  Call Extruder(0.094)
  MoveL 4443 to (501.07, 492.3, 9.5) mm, rotated rx 0 ry 90 rz 0 deg; joints [-11.281, -27.301, 111.303, -15.284, -83.35, 50.807]
  Call Extruder(0.055)
  MoveL 4444 to (501.07, 490.4, 9.5) mm, rotated rx 0 ry 90 rz 0 deg; joints [-11.107, -27.308, 111.347, -15.107, -83.382, 50.779]
  Call Extruder(0.248)
  MoveL 4445 to (509.6, 490.4, 9.5) mm, rotated rx 0 ry 90 rz 0 deg; joints [-10.955, -27.148, 110.323, -14.982, -82.543, 50.989]
  Call Extruder(0.228)
  MoveL 4446 to (509.6, 498.23, 9.5) mm, rotated rx 0 ry 90 rz 0 deg; joints [-11.664, -27.118, 110.135, -15.702, -82.413, 51.114]
  Call Extruder(0.043)
  MoveL 4447 to (508.13, 498.23, 9.5) mm, rotated rx 0 ry 90 rz 0 deg; joints [-11.692, -27.146, 110.312, -15.725, -82.557, 51.076]
  Call Extruder(0.014)
  MoveL 4448 to (507.66, 498.23, 9.5) mm, rotated rx 0 ry 90 rz 0 deg; joints [-11.701, -27.155, 110.368, -15.733, -82.602, 51.065]
  Call Extruder(0.080)
  MoveL 4449 to (507.66, 500.97, 9.5) mm, rotated rx 0 ry 90 rz 0 deg; joints [-11.949, -27.144, 110.299, -15.985, -82.555, 51.109]
  Set speed (120.0 mm/s)
  MoveL 4450 to (508.06, 500.97, 9.5) mm, rotated rx 0 ry 90 rz 0 deg; joints [-11.941, -27.137, 110.251, -15.978, -82.516, 51.119]
  Set speed (1000.0 mm/s)
  MoveL 4451 to (508.06, 501.67, 9.5) mm, rotated rx 0 ry 90 rz 0 deg; joints [-12.005, -27.134, 110.233, -16.043, -82.504, 51.131]
  Set speed (1000.0 mm/s)
  MoveL 4452 to (490.68, 490.68, 9.5) mm, rotated rx 0 ry 90 rz 0 deg; joints [-11.324, -27.485, 112.575, -15.296, -84.401, 50.522]
  Set speed (1000.0 mm/s)
  MoveL 4453 to (490.68, 490.68, 9.6) mm, rotated rx 0 ry 90 rz 0 deg; joints [-11.324, -27.496, 112.58, -15.296, -84.396, 50.523]
  Set speed (30.0 mm/s)
  Call Extruder(0.767)
  MoveL 4454 to (509.32, 509.32, 9.6) mm, rotated rx 0 ry 90 rz 0 deg; joints [-12.669, -27.086, 109.886, -16.723, -82.239, 51.295]
  MoveL 4455 to (509.44, 509.44, 9.6) mm, rotated rx 0 ry 90 rz 0 deg; joints [-12.677, -27.083, 109.868, -16.733, -82.225, 51.301]
  Set speed (120.0 mm/s)
  MoveL 4456 to (508.59, 501.31, 9.6) mm, rotated rx 0 ry 90 rz 0 deg; joints [-11.962, -27.135, 110.184, -16.001, -82.453, 51.14]
  Set speed (30.0 mm/s)
  Call Extruder(0.330)
  MoveL 4457 to (500.58, 509.32, 9.6) mm, rotated rx 0 ry 90 rz 0 deg; joints [-12.847, -27.254, 110.932, -16.871, -83.085, 51.06]
  Set speed (120.0 mm/s)
  MoveL 4458 to (499.42, 509.32, 9.6) mm, rotated rx 0 ry 90 rz 0 deg; joints [-12.872, -27.276, 111.07, -16.891, -83.198, 51.028]
  Set speed (30.0 mm/s)
  Call Extruder(0.360)
  MoveL 4459 to (490.68, 500.58, 9.6) mm, rotated rx 0 ry 90 rz 0 deg; joints [-12.247, -27.462, 112.336, -16.229, -84.216, 50.659]
  Set speed (120.0 mm/s)
  MoveL 4460 to (490.68, 499.42, 9.6) mm, rotated rx 0 ry 90 rz 0 deg; joints [-12.139, -27.466, 112.366, -16.12, -84.237, 50.642]
  Set speed (30.0 mm/s)
  Call Extruder(0.286)
  MoveL 4461 to (497.63, 492.47, 9.6) mm, rotated rx 0 ry 90 rz 0 deg; joints [-11.361, -27.372, 111.714, -15.354, -83.68, 50.724]
  MoveL 4462 to (497.75, 492.35, 9.6) mm, rotated rx 0 ry 90 rz 0 deg; joints [-11.347, -27.371, 111.702, -15.34, -83.67, 50.726]
  Set speed (120.0 mm/s)
  MoveL 4463 to (501.03, 492.33, 9.6) mm, rotated rx 0 ry 90 rz 0 deg; joints [-11.285, -27.312, 111.312, -15.287, -83.348, 50.808]
  Set speed (1000.0 mm/s)
  MoveL 4464 to (501.28, 491.38, 9.6) mm, rotated rx 0 ry 90 rz 0 deg; joints [-11.193, -27.311, 111.304, -15.196, -83.339, 50.8]
  Set speed (30.0 mm/s)
  Call Extruder(0.268)
  MoveL 4465 to (507.79, 497.89, 9.6) mm, rotated rx 0 ry 90 rz 0 deg; joints [-11.668, -27.165, 110.366, -15.699, -82.59, 51.064]
  MoveL 4466 to (507.91, 498.02, 9.6) mm, rotated rx 0 ry 90 rz 0 deg; joints [-11.676, -27.162, 110.348, -15.709, -82.576, 51.069]
  Set speed (120.0 mm/s)
  MoveL 4467 to (509.32, 490.68, 9.6) mm, rotated rx 0 ry 90 rz 0 deg; joints [-10.985, -27.163, 110.356, -15.012, -82.561, 50.987]
  Set speed (30.0 mm/s)
  Call Extruder(0.767)
  MoveL 4468 to (490.68, 509.32, 9.6) mm, rotated rx 0 ry 90 rz 0 deg; joints [-13.056, -27.429, 112.105, -17.048, -84.046, 50.787]
  MoveL 4469 to (490.56, 509.44, 9.6) mm, rotated rx 0 ry 90 rz 0 deg; joints [-13.07, -27.431, 112.116, -17.062, -84.056, 50.785]
  Set speed (120.0 mm/s)
  MoveL 4470 to (507.59, 501.1, 9.6) mm, rotated rx 0 ry 90 rz 0 deg; joints [-11.962, -27.156, 110.31, -15.997, -82.554, 51.111]
  Set speed (1000.0 mm/s)
  MoveL 4471 to (507.66, 501.03, 9.6) mm, rotated rx 0 ry 90 rz 0 deg; joints [-11.954, -27.155, 110.303, -15.99, -82.549, 51.111]
  Set speed (15.0 mm/s)
  Call Extruder(0.056)
  MoveL 4472 to (509.6, 501.03, 9.6) mm, rotated rx 0 ry 90 rz 0 deg; joints [-11.917, -27.117, 110.069, -15.96, -82.36, 51.161]
  Call Extruder(0.249)
  MoveL 4473 to (509.6, 509.6, 9.6) mm, rotated rx 0 ry 90 rz 0 deg; joints [-12.688, -27.079, 109.845, -16.744, -82.206, 51.308]
  Call Extruder(0.559)
  MoveL 4474 to (490.4, 509.6, 9.6) mm, rotated rx 0 ry 90 rz 0 deg; joints [-13.088, -27.433, 112.13, -17.079, -84.068, 50.783]
  MoveL 4475 to (490.4, 490.4, 9.6) mm, rotated rx 0 ry 90 rz 0 deg; joints [-11.303, -27.501, 112.62, -15.274, -84.428, 50.513]
  Call Extruder(0.218)
  MoveL 4476 to (497.9, 490.4, 9.6) mm, rotated rx 0 ry 90 rz 0 deg; joints [-11.164, -27.375, 111.731, -15.156, -83.688, 50.702]
  Call Extruder(0.039)
  MoveL 4477 to (497.9, 491.75, 9.6) mm, rotated rx 0 ry 90 rz 0 deg; joints [-11.289, -27.37, 111.699, -15.282, -83.666, 50.721]
  Call Extruder(0.016)
  MoveL 4478 to (497.91, 492.3, 9.6) mm, rotated rx 0 ry 90 rz 0 deg; joints [-11.34, -27.368, 111.685, -15.333, -83.655, 50.729]
  Call Extruder(0.090)
  MoveL 4479 to (501, 492.3, 9.6) mm, rotated rx 0 ry 90 rz 0 deg; joints [-11.283, -27.313, 111.316, -15.285, -83.351, 50.807]
  Call Extruder(0.055)
  MoveL 4480 to (501.01, 490.4, 9.6) mm, rotated rx 0 ry 90 rz 0 deg; joints [-11.108, -27.32, 111.36, -15.108, -83.383, 50.779]
  Call Extruder(0.250)
  MoveL 4481 to (509.6, 490.4, 9.6) mm, rotated rx 0 ry 90 rz 0 deg; joints [-10.955, -27.159, 110.329, -14.982, -82.538, 50.99]
  Call Extruder(0.226)
  MoveL 4482 to (509.6, 498.17, 9.6) mm, rotated rx 0 ry 90 rz 0 deg; joints [-11.659, -27.128, 110.141, -15.697, -82.409, 51.114]
  Call Extruder(0.056)
  MoveL 4483 to (507.66, 498.17, 9.6) mm, rotated rx 0 ry 90 rz 0 deg; joints [-11.695, -27.166, 110.374, -15.727, -82.598, 51.065]
  Call Extruder(0.083)
  MoveL 4484 to (507.66, 501.03, 9.6) mm, rotated rx 0 ry 90 rz 0 deg; joints [-11.954, -27.155, 110.303, -15.99, -82.549, 51.111]
  Set speed (120.0 mm/s)
  MoveL 4485 to (508.06, 501.03, 9.6) mm, rotated rx 0 ry 90 rz 0 deg; joints [-11.947, -27.147, 110.255, -15.984, -82.51, 51.122]
  Set speed (1000.0 mm/s)
  MoveL 4486 to (508.06, 501.73, 9.6) mm, rotated rx 0 ry 90 rz 0 deg; joints [-12.01, -27.144, 110.237, -16.048, -82.497, 51.133]
  Set speed (1000.0 mm/s)
  MoveL 4487 to (490.68, 490.68, 9.6) mm, rotated rx 0 ry 90 rz 0 deg; joints [-11.324, -27.496, 112.58, -15.296, -84.396, 50.523]
  Set speed (1000.0 mm/s)
  MoveL 4488 to (490.68, 490.68, 9.7) mm, rotated rx 0 ry 90 rz 0 deg; joints [-11.324, -27.506, 112.585, -15.296, -84.391, 50.525]
  Set speed (30.0 mm/s)
  Call Extruder(0.767)
  MoveL 4489 to (509.32, 509.32, 9.7) mm, rotated rx 0 ry 90 rz 0 deg; joints [-12.669, -27.097, 109.891, -16.724, -82.234, 51.297]
  MoveL 4490 to (509.44, 509.44, 9.7) mm, rotated rx 0 ry 90 rz 0 deg; joints [-12.677, -27.094, 109.873, -16.733, -82.22, 51.302]
  Set speed (120.0 mm/s)
  MoveL 4491 to (508.53, 501.37, 9.7) mm, rotated rx 0 ry 90 rz 0 deg; joints [-11.968, -27.147, 110.195, -16.007, -82.453, 51.141]
  Set speed (30.0 mm/s)
  Call Extruder(0.327)
  MoveL 4492 to (500.58, 509.32, 9.7) mm, rotated rx 0 ry 90 rz 0 deg; joints [-12.847, -27.265, 110.937, -16.871, -83.08, 51.061]
  Set speed (120.0 mm/s)
  MoveL 4493 to (499.42, 509.32, 9.7) mm, rotated rx 0 ry 90 rz 0 deg; joints [-12.872, -27.286, 111.075, -16.891, -83.193, 51.03]
  Set speed (30.0 mm/s)
  Call Extruder(0.360)
  MoveL 4494 to (490.68, 500.58, 9.7) mm, rotated rx 0 ry 90 rz 0 deg; joints [-12.247, -27.472, 112.342, -16.229, -84.21, 50.66]
  Set speed (120.0 mm/s)
  MoveL 4495 to (490.68, 499.42, 9.7) mm, rotated rx 0 ry 90 rz 0 deg; joints [-12.139, -27.477, 112.371, -16.12, -84.232, 50.644]
  Set speed (30.0 mm/s)
  Call Extruder(0.288)
  MoveL 4496 to (497.68, 492.42, 9.7) mm, rotated rx 0 ry 90 rz 0 deg; joints [-11.355, -27.382, 111.714, -15.348, -83.671, 50.726]
  MoveL 4497 to (497.8, 492.3, 9.7) mm, rotated rx 0 ry 90 rz 0 deg; joints [-11.342, -27.381, 111.703, -15.335, -83.661, 50.728]
  Set speed (120.0 mm/s)
  MoveL 4498 to (500.97, 492.33, 9.7) mm, rotated rx 0 ry 90 rz 0 deg; joints [-11.286, -27.324, 111.324, -15.289, -83.349, 50.808]
  Set speed (1000.0 mm/s)
  MoveL 4499 to (501.22, 491.32, 9.7) mm, rotated rx 0 ry 90 rz 0 deg; joints [-11.189, -27.323, 111.318, -15.191, -83.341, 50.799]
  Set speed (30.0 mm/s)
  Call Extruder(0.268)
  MoveL 4500 to (507.73, 497.83, 9.7) mm, rotated rx 0 ry 90 rz 0 deg; joints [-11.663, -27.177, 110.38, -15.695, -82.592, 51.063]
  MoveL 4501 to (507.85, 497.95, 9.7) mm, rotated rx 0 ry 90 rz 0 deg; joints [-11.672, -27.174, 110.362, -15.704, -82.578, 51.068]
  Set speed (120.0 mm/s)
  MoveL 4502 to (509.32, 490.68, 9.7) mm, rotated rx 0 ry 90 rz 0 deg; joints [-10.985, -27.174, 110.361, -15.012, -82.556, 50.989]
  Set speed (30.0 mm/s)
  Call Extruder(0.767)
  MoveL 4503 to (490.68, 509.32, 9.7) mm, rotated rx 0 ry 90 rz 0 deg; joints [-13.056, -27.44, 112.11, -17.048, -84.041, 50.789]
  MoveL 4504 to (490.56, 509.44, 9.7) mm, rotated rx 0 ry 90 rz 0 deg; joints [-13.07, -27.441, 112.121, -17.062, -84.051, 50.787]
  Set speed (120.0 mm/s)
  MoveL 4505 to (501.01, 492.37, 9.7) mm, rotated rx 0 ry 90 rz 0 deg; joints [-11.289, -27.323, 111.318, -15.292, -83.344, 50.809]
  Set speed (1000.0 mm/s)
  MoveL 4506 to (500.94, 492.3, 9.7) mm, rotated rx 0 ry 90 rz 0 deg; joints [-11.284, -27.325, 111.328, -15.286, -83.352, 50.806]
  Set speed (15.0 mm/s)
  Call Extruder(0.055)
  MoveL 4507 to (500.94, 490.4, 9.7) mm, rotated rx 0 ry 90 rz 0 deg; joints [-11.109, -27.332, 111.373, -15.109, -83.384, 50.779]
  Call Extruder(0.252)
  MoveL 4508 to (509.6, 490.4, 9.7) mm, rotated rx 0 ry 90 rz 0 deg; joints [-10.955, -27.169, 110.334, -14.982, -82.533, 50.991]
  Call Extruder(0.224)
  MoveL 4509 to (509.6, 498.11, 9.7) mm, rotated rx 0 ry 90 rz 0 deg; joints [-11.653, -27.139, 110.148, -15.692, -82.405, 51.115]
  Call Extruder(0.056)
  MoveL 4510 to (507.66, 498.11, 9.7) mm, rotated rx 0 ry 90 rz 0 deg; joints [-11.69, -27.177, 110.381, -15.722, -82.594, 51.066]
  Call Extruder(0.087)
  MoveL 4511 to (507.66, 501.09, 9.7) mm, rotated rx 0 ry 90 rz 0 deg; joints [-11.959, -27.165, 110.306, -15.995, -82.542, 51.114]
  Call Extruder(0.056)
  MoveL 4512 to (509.6, 501.09, 9.7) mm, rotated rx 0 ry 90 rz 0 deg; joints [-11.923, -27.127, 110.073, -15.965, -82.353, 51.164]
  Call Extruder(0.248)
  MoveL 4513 to (509.6, 509.6, 9.7) mm, rotated rx 0 ry 90 rz 0 deg; joints [-12.688, -27.09, 109.85, -16.745, -82.201, 51.309]
  Call Extruder(0.559)
  MoveL 4514 to (490.4, 509.6, 9.7) mm, rotated rx 0 ry 90 rz 0 deg; joints [-13.088, -27.443, 112.135, -17.079, -84.063, 50.785]
  MoveL 4515 to (490.4, 490.4, 9.7) mm, rotated rx 0 ry 90 rz 0 deg; joints [-11.303, -27.512, 112.625, -15.274, -84.423, 50.514]
  Call Extruder(0.220)
  MoveL 4516 to (497.95, 490.4, 9.7) mm, rotated rx 0 ry 90 rz 0 deg; joints [-11.163, -27.385, 111.729, -15.155, -83.678, 50.704]
  Call Extruder(0.055)
  MoveL 4517 to (497.96, 492.3, 9.7) mm, rotated rx 0 ry 90 rz 0 deg; joints [-11.339, -27.378, 111.684, -15.332, -83.645, 50.732]
  Call Extruder(0.087)
  MoveL 4518 to (500.94, 492.3, 9.7) mm, rotated rx 0 ry 90 rz 0 deg; joints [-11.284, -27.325, 111.328, -15.286, -83.352, 50.806]
  Set speed (120.0 mm/s)
  MoveL 4519 to (500.94, 491.9, 9.7) mm, rotated rx 0 ry 90 rz 0 deg; joints [-11.247, -27.326, 111.338, -15.249, -83.359, 50.801]
  Set speed (1000.0 mm/s)
  MoveL 4520 to (501.64, 491.9, 9.7) mm, rotated rx 0 ry 90 rz 0 deg; joints [-11.234, -27.314, 111.254, -15.238, -83.29, 50.818]
  Set speed (1000.0 mm/s)
  MoveL 4521 to (497.93, 492.32, 9.7) mm, rotated rx 0 ry 90 rz 0 deg; joints [-11.342, -27.378, 111.686, -15.336, -83.647, 50.731]
  Set speed (1000.0 mm/s)
  MoveL 4522 to (490.68, 490.68, 9.7) mm, rotated rx 0 ry 90 rz 0 deg; joints [-11.324, -27.506, 112.585, -15.296, -84.391, 50.525]
  Set speed (1000.0 mm/s)
  MoveL 4523 to (490.68, 490.68, 9.8) mm, rotated rx 0 ry 90 rz 0 deg; joints [-11.324, -27.517, 112.591, -15.296, -84.385, 50.526]
  Set speed (30.0 mm/s)
  Call Extruder(0.767)
  MoveL 4524 to (509.32, 509.32, 9.8) mm, rotated rx 0 ry 90 rz 0 deg; joints [-12.669, -27.107, 109.896, -16.724, -82.229, 51.298]
  MoveL 4525 to (509.44, 509.44, 9.8) mm, rotated rx 0 ry 90 rz 0 deg; joints [-12.677, -27.104, 109.878, -16.733, -82.214, 51.304]
  Set speed (120.0 mm/s)
  MoveL 4526 to (508.47, 501.42, 9.8) mm, rotated rx 0 ry 90 rz 0 deg; joints [-11.974, -27.158, 110.205, -16.014, -82.452, 51.142]
  Set speed (30.0 mm/s)
  Call Extruder(0.325)
  MoveL 4527 to (500.58, 509.32, 9.8) mm, rotated rx 0 ry 90 rz 0 deg; joints [-12.847, -27.275, 110.943, -16.871, -83.075, 51.063]
  Set speed (120.0 mm/s)
  MoveL 4528 to (499.42, 509.32, 9.8) mm, rotated rx 0 ry 90 rz 0 deg; joints [-12.872, -27.297, 111.081, -16.891, -83.188, 51.031]
  Set speed (30.0 mm/s)
  Call Extruder(0.360)
  MoveL 4529 to (490.68, 500.58, 9.8) mm, rotated rx 0 ry 90 rz 0 deg; joints [-12.247, -27.483, 112.347, -16.229, -84.205, 50.662]
  Set speed (120.0 mm/s)
  MoveL 4530 to (490.68, 499.42, 9.8) mm, rotated rx 0 ry 90 rz 0 deg; joints [-12.139, -27.487, 112.376, -16.12, -84.227, 50.645]
  Set speed (30.0 mm/s)
  Call Extruder(0.290)
  MoveL 4531 to (497.73, 492.36, 9.8) mm, rotated rx 0 ry 90 rz 0 deg; joints [-11.349, -27.392, 111.714, -15.342, -83.661, 50.728]
  MoveL 4532 to (497.86, 492.24, 9.8) mm, rotated rx 0 ry 90 rz 0 deg; joints [-11.335, -27.39, 111.702, -15.329, -83.651, 50.73]
  Set speed (120.0 mm/s)
  MoveL 4533 to (500.9, 492.32, 9.8) mm, rotated rx 0 ry 90 rz 0 deg; joints [-11.287, -27.336, 111.337, -15.29, -83.35, 50.807]
  Set speed (1000.0 mm/s)
  MoveL 4534 to (501.16, 491.26, 9.8) mm, rotated rx 0 ry 90 rz 0 deg; joints [-11.184, -27.335, 111.332, -15.186, -83.343, 50.798]
  Set speed (30.0 mm/s)
  Call Extruder(0.268)
  MoveL 4535 to (507.67, 497.77, 9.8) mm, rotated rx 0 ry 90 rz 0 deg; joints [-11.659, -27.189, 110.394, -15.69, -82.594, 51.062]
  MoveL 4536 to (507.79, 497.89, 9.8) mm, rotated rx 0 ry 90 rz 0 deg; joints [-11.668, -27.186, 110.376, -15.7, -82.58, 51.067]
  Set speed (120.0 mm/s)
  MoveL 4537 to (509.32, 490.68, 9.8) mm, rotated rx 0 ry 90 rz 0 deg; joints [-10.985, -27.184, 110.366, -15.012, -82.55, 50.99]
  Set speed (30.0 mm/s)
  Call Extruder(0.767)
  MoveL 4538 to (490.68, 509.32, 9.8) mm, rotated rx 0 ry 90 rz 0 deg; joints [-13.056, -27.45, 112.115, -17.048, -84.036, 50.79]
  MoveL 4539 to (490.56, 509.44, 9.8) mm, rotated rx 0 ry 90 rz 0 deg; joints [-13.07, -27.452, 112.127, -17.062, -84.046, 50.789]
  Set speed (120.0 mm/s)
  MoveL 4540 to (500.95, 492.37, 9.8) mm, rotated rx 0 ry 90 rz 0 deg; joints [-11.29, -27.335, 111.331, -15.293, -83.345, 50.809]
  Set speed (1000.0 mm/s)
  MoveL 4541 to (500.88, 492.3, 9.8) mm, rotated rx 0 ry 90 rz 0 deg; joints [-11.285, -27.336, 111.341, -15.287, -83.353, 50.806]
  Set speed (15.0 mm/s)
  Call Extruder(0.055)
  MoveL 4542 to (500.88, 490.4, 9.8) mm, rotated rx 0 ry 90 rz 0 deg; joints [-11.11, -27.343, 111.386, -15.111, -83.385, 50.779]
  Call Extruder(0.254)
  MoveL 4543 to (509.6, 490.4, 9.8) mm, rotated rx 0 ry 90 rz 0 deg; joints [-10.955, -27.18, 110.339, -14.982, -82.527, 50.993]
  Call Extruder(0.223)
  MoveL 4544 to (509.6, 498.05, 9.8) mm, rotated rx 0 ry 90 rz 0 deg; joints [-11.648, -27.15, 110.155, -15.686, -82.401, 51.115]
  Call Extruder(0.056)
  MoveL 4545 to (507.66, 498.05, 9.8) mm, rotated rx 0 ry 90 rz 0 deg; joints [-11.684, -27.188, 110.388, -15.716, -82.59, 51.066]
  Call Extruder(0.090)
  MoveL 4546 to (507.66, 501.14, 9.8) mm, rotated rx 0 ry 90 rz 0 deg; joints [-11.964, -27.175, 110.31, -16.001, -82.536, 51.116]
  Call Extruder(0.056)
  MoveL 4547 to (509.6, 501.15, 9.8) mm, rotated rx 0 ry 90 rz 0 deg; joints [-11.928, -27.137, 110.077, -15.971, -82.347, 51.166]
  Call Extruder(0.246)
  MoveL 4548 to (509.6, 509.6, 9.8) mm, rotated rx 0 ry 90 rz 0 deg; joints [-12.688, -27.1, 109.855, -16.745, -82.196, 51.311]
  Call Extruder(0.559)
  MoveL 4549 to (490.4, 509.6, 9.8) mm, rotated rx 0 ry 90 rz 0 deg; joints [-13.088, -27.454, 112.141, -17.08, -84.058, 50.787]
  MoveL 4550 to (490.4, 490.4, 9.8) mm, rotated rx 0 ry 90 rz 0 deg; joints [-11.303, -27.522, 112.63, -15.274, -84.418, 50.515]
  Call Extruder(0.221)
  MoveL 4551 to (498.01, 490.4, 9.8) mm, rotated rx 0 ry 90 rz 0 deg; joints [-11.162, -27.394, 111.728, -15.154, -83.667, 50.707]
  Call Extruder(0.055)
  MoveL 4552 to (498.02, 492.3, 9.8) mm, rotated rx 0 ry 90 rz 0 deg; joints [-11.338, -27.387, 111.682, -15.332, -83.634, 50.734]
  Call Extruder(0.083)
  MoveL 4553 to (500.88, 492.3, 9.8) mm, rotated rx 0 ry 90 rz 0 deg; joints [-11.285, -27.336, 111.341, -15.287, -83.353, 50.806]
  Set speed (120.0 mm/s)
  MoveL 4554 to (500.88, 491.9, 9.8) mm, rotated rx 0 ry 90 rz 0 deg; joints [-11.248, -27.338, 111.351, -15.25, -83.36, 50.8]
  Set speed (1000.0 mm/s)
  MoveL 4555 to (501.58, 491.9, 9.8) mm, rotated rx 0 ry 90 rz 0 deg; joints [-11.235, -27.325, 111.267, -15.239, -83.291, 50.818]
  Set speed (1000.0 mm/s)
  MoveL 4556 to (497.99, 492.33, 9.8) mm, rotated rx 0 ry 90 rz 0 deg; joints [-11.341, -27.388, 111.685, -15.335, -83.636, 50.734]
  Set speed (1000.0 mm/s)
  MoveL 4557 to (490.68, 490.68, 9.8) mm, rotated rx 0 ry 90 rz 0 deg; joints [-11.324, -27.517, 112.591, -15.296, -84.385, 50.526]
  Set speed (1000.0 mm/s)
  MoveL 4558 to (490.68, 490.68, 9.9) mm, rotated rx 0 ry 90 rz 0 deg; joints [-11.324, -27.528, 112.596, -15.296, -84.38, 50.528]
  Set speed (30.0 mm/s)
  Call Extruder(0.767)
  MoveL 4559 to (509.32, 509.32, 9.9) mm, rotated rx 0 ry 90 rz 0 deg; joints [-12.669, -27.118, 109.902, -16.724, -82.224, 51.3]
  MoveL 4560 to (509.44, 509.44, 9.9) mm, rotated rx 0 ry 90 rz 0 deg; joints [-12.677, -27.115, 109.883, -16.733, -82.209, 51.305]
  Set speed (120.0 mm/s)
  MoveL 4561 to (508.42, 501.48, 9.9) mm, rotated rx 0 ry 90 rz 0 deg; joints [-11.98, -27.169, 110.216, -16.02, -82.452, 51.143]
  Set speed (30.0 mm/s)
  Call Extruder(0.323)
  MoveL 4562 to (500.58, 509.32, 9.9) mm, rotated rx 0 ry 90 rz 0 deg; joints [-12.847, -27.286, 110.948, -16.871, -83.07, 51.064]
  Set speed (120.0 mm/s)
  MoveL 4563 to (499.42, 509.32, 9.9) mm, rotated rx 0 ry 90 rz 0 deg; joints [-12.872, -27.307, 111.086, -16.892, -83.183, 51.033]
  Set speed (30.0 mm/s)
  Call Extruder(0.360)
  MoveL 4564 to (490.68, 500.58, 9.9) mm, rotated rx 0 ry 90 rz 0 deg; joints [-12.247, -27.494, 112.352, -16.229, -84.2, 50.663]
  Set speed (120.0 mm/s)
  MoveL 4565 to (490.68, 499.42, 9.9) mm, rotated rx 0 ry 90 rz 0 deg; joints [-12.139, -27.498, 112.382, -16.12, -84.222, 50.647]
  Set speed (30.0 mm/s)
  Call Extruder(0.293)
  MoveL 4566 to (497.79, 492.31, 9.9) mm, rotated rx 0 ry 90 rz 0 deg; joints [-11.343, -27.402, 111.714, -15.336, -83.651, 50.73]
  MoveL 4567 to (497.91, 492.18, 9.9) mm, rotated rx 0 ry 90 rz 0 deg; joints [-11.329, -27.4, 111.702, -15.323, -83.641, 50.732]
  Set speed (120.0 mm/s)
  MoveL 4568 to (500.84, 492.32, 9.9) mm, rotated rx 0 ry 90 rz 0 deg; joints [-11.288, -27.348, 111.35, -15.291, -83.351, 50.807]
  Set speed (1000.0 mm/s)
  MoveL 4569 to (501.09, 491.19, 9.9) mm, rotated rx 0 ry 90 rz 0 deg; joints [-11.179, -27.347, 111.347, -15.181, -83.345, 50.797]
  Set speed (30.0 mm/s)
  Call Extruder(0.268)
  MoveL 4570 to (507.61, 497.71, 9.9) mm, rotated rx 0 ry 90 rz 0 deg; joints [-11.654, -27.2, 110.408, -15.686, -82.596, 51.061]
  MoveL 4571 to (507.73, 497.83, 9.9) mm, rotated rx 0 ry 90 rz 0 deg; joints [-11.663, -27.198, 110.39, -15.695, -82.582, 51.066]
  Set speed (120.0 mm/s)
  MoveL 4572 to (509.32, 490.68, 9.9) mm, rotated rx 0 ry 90 rz 0 deg; joints [-10.985, -27.195, 110.372, -15.012, -82.545, 50.992]
  Set speed (30.0 mm/s)
  Call Extruder(0.767)
  MoveL 4573 to (490.68, 509.32, 9.9) mm, rotated rx 0 ry 90 rz 0 deg; joints [-13.056, -27.461, 112.121, -17.048, -84.031, 50.792]
  MoveL 4574 to (490.56, 509.44, 9.9) mm, rotated rx 0 ry 90 rz 0 deg; joints [-13.07, -27.463, 112.132, -17.062, -84.04, 50.79]
  Set speed (120.0 mm/s)
  MoveL 4575 to (500.88, 492.37, 9.9) mm, rotated rx 0 ry 90 rz 0 deg; joints [-11.291, -27.347, 111.344, -15.294, -83.346, 50.809]
  Set speed (1000.0 mm/s)
  MoveL 4576 to (500.81, 492.3, 9.9) mm, rotated rx 0 ry 90 rz 0 deg; joints [-11.286, -27.348, 111.354, -15.289, -83.354, 50.806]
  Set speed (15.0 mm/s)
  Call Extruder(0.055)
  MoveL 4577 to (500.82, 490.4, 9.9) mm, rotated rx 0 ry 90 rz 0 deg; joints [-11.112, -27.355, 111.398, -15.112, -83.386, 50.778]
  Call Extruder(0.256)
  MoveL 4578 to (509.6, 490.4, 9.9) mm, rotated rx 0 ry 90 rz 0 deg; joints [-10.955, -27.19, 110.344, -14.983, -82.522, 50.994]
  Call Extruder(0.221)
  MoveL 4579 to (509.6, 497.99, 9.9) mm, rotated rx 0 ry 90 rz 0 deg; joints [-11.643, -27.16, 110.162, -15.681, -82.397, 51.116]
  Call Extruder(0.056)
  MoveL 4580 to (507.66, 497.99, 9.9) mm, rotated rx 0 ry 90 rz 0 deg; joints [-11.679, -27.198, 110.394, -15.711, -82.586, 51.067]
  Call Extruder(0.093)
  MoveL 4581 to (507.66, 501.2, 9.9) mm, rotated rx 0 ry 90 rz 0 deg; joints [-11.97, -27.185, 110.314, -16.006, -82.53, 51.119]
  Call Extruder(0.056)
  MoveL 4582 to (509.6, 501.2, 9.9) mm, rotated rx 0 ry 90 rz 0 deg; joints [-11.933, -27.147, 110.081, -15.976, -82.341, 51.169]
  Call Extruder(0.244)
  MoveL 4583 to (509.6, 509.6, 9.9) mm, rotated rx 0 ry 90 rz 0 deg; joints [-12.688, -27.111, 109.86, -16.745, -82.191, 51.312]
  Call Extruder(0.559)
  MoveL 4584 to (490.4, 509.6, 9.9) mm, rotated rx 0 ry 90 rz 0 deg; joints [-13.088, -27.465, 112.146, -17.08, -84.052, 50.788]
  MoveL 4585 to (490.4, 490.4, 9.9) mm, rotated rx 0 ry 90 rz 0 deg; joints [-11.303, -27.533, 112.636, -15.275, -84.413, 50.517]
  Call Extruder(0.223)
  MoveL 4586 to (498.07, 490.4, 9.9) mm, rotated rx 0 ry 90 rz 0 deg; joints [-11.161, -27.404, 111.726, -15.154, -83.656, 50.71]
  Call Extruder(0.042)
  MoveL 4587 to (498.07, 491.84, 9.9) mm, rotated rx 0 ry 90 rz 0 deg; joints [-11.294, -27.399, 111.692, -15.288, -83.632, 50.73]
  Call Extruder(0.013)
  MoveL 4588 to (498.07, 492.3, 9.9) mm, rotated rx 0 ry 90 rz 0 deg; joints [-11.337, -27.397, 111.681, -15.331, -83.623, 50.737]
  Call Extruder(0.080)
  MoveL 4589 to (500.81, 492.3, 9.9) mm, rotated rx 0 ry 90 rz 0 deg; joints [-11.286, -27.348, 111.354, -15.289, -83.354, 50.806]
  Set speed (120.0 mm/s)
  MoveL 4590 to (500.81, 491.9, 9.9) mm, rotated rx 0 ry 90 rz 0 deg; joints [-11.249, -27.35, 111.363, -15.251, -83.361, 50.8]
  Set speed (1000.0 mm/s)
  MoveL 4591 to (501.51, 491.9, 9.9) mm, rotated rx 0 ry 90 rz 0 deg; joints [-11.237, -27.337, 111.28, -15.241, -83.292, 50.818]
  Set speed (1000.0 mm/s)
  MoveL 4592 to (498.04, 492.33, 9.9) mm, rotated rx 0 ry 90 rz 0 deg; joints [-11.34, -27.397, 111.683, -15.334, -83.626, 50.737]
  Set speed (1000.0 mm/s)
  MoveL 4593 to (490.68, 490.68, 9.9) mm, rotated rx 0 ry 90 rz 0 deg; joints [-11.324, -27.528, 112.596, -15.296, -84.38, 50.528]
  Set speed (1000.0 mm/s)
  MoveL 4594 to (490.68, 490.68, 10) mm, rotated rx 0 ry 90 rz 0 deg; joints [-11.324, -27.538, 112.601, -15.297, -84.375, 50.529]
  Set speed (30.0 mm/s)
  Call Extruder(0.767)
  MoveL 4595 to (509.32, 509.32, 10) mm, rotated rx 0 ry 90 rz 0 deg; joints [-12.669, -27.128, 109.907, -16.724, -82.219, 51.301]
  MoveL 4596 to (509.44, 509.44, 10) mm, rotated rx 0 ry 90 rz 0 deg; joints [-12.677, -27.125, 109.889, -16.733, -82.204, 51.307]
  Set speed (120.0 mm/s)
  MoveL 4597 to (508.36, 501.54, 10) mm, rotated rx 0 ry 90 rz 0 deg; joints [-11.987, -27.181, 110.227, -16.026, -82.451, 51.144]
  Set speed (30.0 mm/s)
  Call Extruder(0.320)
  MoveL 4598 to (500.58, 509.32, 10) mm, rotated rx 0 ry 90 rz 0 deg; joints [-12.847, -27.296, 110.953, -16.872, -83.065, 51.066]
  Set speed (120.0 mm/s)
  MoveL 4599 to (499.42, 509.32, 10) mm, rotated rx 0 ry 90 rz 0 deg; joints [-12.872, -27.318, 111.091, -16.892, -83.177, 51.034]
  Set speed (30.0 mm/s)
  Call Extruder(0.360)
  MoveL 4600 to (490.68, 500.58, 10) mm, rotated rx 0 ry 90 rz 0 deg; joints [-12.247, -27.504, 112.357, -16.229, -84.195, 50.665]
  Set speed (120.0 mm/s)
  MoveL 4601 to (490.68, 499.42, 10) mm, rotated rx 0 ry 90 rz 0 deg; joints [-12.139, -27.508, 112.387, -16.12, -84.217, 50.648]
  Set speed (30.0 mm/s)
  Call Extruder(0.297)
  MoveL 4602 to (497.91, 492.19, 10) mm, rotated rx 0 ry 90 rz 0 deg; joints [-11.33, -27.411, 111.708, -15.324, -83.637, 50.733]
  MoveL 4603 to (498.03, 492.07, 10) mm, rotated rx 0 ry 90 rz 0 deg; joints [-11.316, -27.409, 111.697, -15.311, -83.627, 50.734]
  Set speed (120.0 mm/s)
  MoveL 4604 to (500.32, 492.34, 10) mm, rotated rx 0 ry 90 rz 0 deg; joints [-11.299, -27.367, 111.417, -15.3, -83.396, 50.796]
  Set speed (1000.0 mm/s)
  MoveL 4605 to (501.03, 491.13, 10) mm, rotated rx 0 ry 90 rz 0 deg; joints [-11.175, -27.359, 111.361, -15.177, -83.347, 50.796]
  Set speed (30.0 mm/s)
  Call Extruder(0.268)
  MoveL 4606 to (507.55, 497.65, 10) mm, rotated rx 0 ry 90 rz 0 deg; joints [-11.65, -27.212, 110.421, -15.682, -82.597, 51.06]
  MoveL 4607 to (507.68, 497.78, 10) mm, rotated rx 0 ry 90 rz 0 deg; joints [-11.659, -27.209, 110.404, -15.691, -82.583, 51.065]
  Set speed (120.0 mm/s)
  MoveL 4608 to (509.32, 490.68, 10) mm, rotated rx 0 ry 90 rz 0 deg; joints [-10.985, -27.205, 110.377, -15.012, -82.54, 50.993]
  Set speed (30.0 mm/s)
  Call Extruder(0.767)
  MoveL 4609 to (490.68, 509.32, 10) mm, rotated rx 0 ry 90 rz 0 deg; joints [-13.056, -27.472, 112.126, -17.048, -84.026, 50.793]
  MoveL 4610 to (490.56, 509.44, 10) mm, rotated rx 0 ry 90 rz 0 deg; joints [-13.07, -27.473, 112.137, -17.062, -84.035, 50.792]
  Set speed (120.0 mm/s)
  MoveL 4611 to (507.59, 501.33, 10) mm, rotated rx 0 ry 90 rz 0 deg; joints [-11.982, -27.197, 110.324, -16.019, -82.53, 51.12]
  Set speed (1000.0 mm/s)
  MoveL 4612 to (507.66, 501.25, 10) mm, rotated rx 0 ry 90 rz 0 deg; joints [-11.975, -27.196, 110.318, -16.011, -82.524, 51.121]
  Set speed (15.0 mm/s)
  Call Extruder(0.056)
  MoveL 4613 to (509.6, 501.26, 10) mm, rotated rx 0 ry 90 rz 0 deg; joints [-11.938, -27.157, 110.084, -15.982, -82.335, 51.171]
  Call Extruder(0.243)
  MoveL 4614 to (509.6, 509.6, 10) mm, rotated rx 0 ry 90 rz 0 deg; joints [-12.688, -27.121, 109.865, -16.745, -82.186, 51.314]
  Call Extruder(0.559)
  MoveL 4615 to (490.4, 509.6, 10) mm, rotated rx 0 ry 90 rz 0 deg; joints [-13.088, -27.475, 112.151, -17.08, -84.047, 50.79]
  MoveL 4616 to (490.4, 490.4, 10) mm, rotated rx 0 ry 90 rz 0 deg; joints [-11.303, -27.544, 112.641, -15.275, -84.407, 50.518]
  Call Extruder(0.225)
  MoveL 4617 to (498.12, 490.4, 10) mm, rotated rx 0 ry 90 rz 0 deg; joints [-11.16, -27.413, 111.725, -15.153, -83.646, 50.713]
  Call Extruder(0.047)
  MoveL 4618 to (498.12, 492.01, 10) mm, rotated rx 0 ry 90 rz 0 deg; joints [-11.31, -27.408, 111.687, -15.304, -83.618, 50.736]
  Call Extruder(0.011)
  MoveL 4619 to (498.37, 492.3, 10) mm, rotated rx 0 ry 90 rz 0 deg; joints [-11.331, -27.402, 111.65, -15.327, -83.589, 50.746]
  Call Extruder(0.057)
  MoveL 4620 to (500.32, 492.3, 10) mm, rotated rx 0 ry 90 rz 0 deg; joints [-11.295, -27.368, 111.418, -15.296, -83.397, 50.795]
  Call Extruder(0.013)
  MoveL 4621 to (500.75, 492.19, 10) mm, rotated rx 0 ry 90 rz 0 deg; joints [-11.277, -27.36, 111.369, -15.28, -83.357, 50.804]
  Call Extruder(0.052)
  MoveL 4622 to (500.75, 490.4, 10) mm, rotated rx 0 ry 90 rz 0 deg; joints [-11.113, -27.367, 111.411, -15.113, -83.387, 50.778]
  Call Extruder(0.258)
  MoveL 4623 to (509.6, 490.4, 10) mm, rotated rx 0 ry 90 rz 0 deg; joints [-10.955, -27.201, 110.349, -14.983, -82.517, 50.995]
  Call Extruder(0.219)
  MoveL 4624 to (509.6, 497.93, 10) mm, rotated rx 0 ry 90 rz 0 deg; joints [-11.637, -27.171, 110.168, -15.676, -82.393, 51.116]
  Call Extruder(0.056)
  MoveL 4625 to (507.66, 497.93, 10) mm, rotated rx 0 ry 90 rz 0 deg; joints [-11.674, -27.209, 110.401, -15.706, -82.582, 51.067]
  Call Extruder(0.097)
  MoveL 4626 to (507.66, 501.25, 10) mm, rotated rx 0 ry 90 rz 0 deg; joints [-11.975, -27.196, 110.318, -16.011, -82.524, 51.121]
  Set speed (120.0 mm/s)
  MoveL 4627 to (508.06, 501.26, 10) mm, rotated rx 0 ry 90 rz 0 deg; joints [-11.967, -27.188, 110.27, -16.005, -82.485, 51.131]
  Set speed (1000.0 mm/s)
  MoveL 4628 to (508.06, 501.96, 10) mm, rotated rx 0 ry 90 rz 0 deg; joints [-12.03, -27.185, 110.252, -16.07, -82.473, 51.143]
  Set speed (1000.0 mm/s)
  MoveL 4629 to (490.68, 490.68, 10) mm, rotated rx 0 ry 90 rz 0 deg; joints [-11.324, -27.538, 112.601, -15.297, -84.375, 50.529]
  Set speed (1000.0 mm/s)
  MoveL 4630 to (490.68, 490.68, 10.1) mm, rotated rx 0 ry 90 rz 0 deg; joints [-11.324, -27.549, 112.606, -15.297, -84.37, 50.531]
  Set speed (30.0 mm/s)
  Call Extruder(0.767)
  MoveL 4631 to (509.32, 509.32, 10.1) mm, rotated rx 0 ry 90 rz 0 deg; joints [-12.669, -27.138, 109.912, -16.724, -82.214, 51.303]
  MoveL 4632 to (509.44, 509.44, 10.1) mm, rotated rx 0 ry 90 rz 0 deg; joints [-12.677, -27.135, 109.894, -16.734, -82.199, 51.308]
  Set speed (120.0 mm/s)
  MoveL 4633 to (508.3, 501.59, 10.1) mm, rotated rx 0 ry 90 rz 0 deg; joints [-11.993, -27.192, 110.237, -16.033, -82.451, 51.145]
  Set speed (30.0 mm/s)
  Call Extruder(0.318)
  MoveL 4634 to (500.58, 509.32, 10.1) mm, rotated rx 0 ry 90 rz 0 deg; joints [-12.847, -27.307, 110.958, -16.872, -83.06, 51.067]
  Set speed (120.0 mm/s)
  MoveL 4635 to (499.42, 509.32, 10.1) mm, rotated rx 0 ry 90 rz 0 deg; joints [-12.872, -27.328, 111.096, -16.892, -83.172, 51.036]
  Set speed (30.0 mm/s)
  Call Extruder(0.360)
  MoveL 4636 to (490.68, 500.58, 10.1) mm, rotated rx 0 ry 90 rz 0 deg; joints [-12.247, -27.515, 112.363, -16.229, -84.19, 50.666]
  Set speed (120.0 mm/s)
  MoveL 4637 to (490.68, 499.42, 10.1) mm, rotated rx 0 ry 90 rz 0 deg; joints [-12.139, -27.519, 112.392, -16.12, -84.211, 50.65]
  Set speed (30.0 mm/s)
  Call Extruder(0.297)
  MoveL 4638 to (497.89, 492.2, 10.1) mm, rotated rx 0 ry 90 rz 0 deg; joints [-11.331, -27.422, 111.714, -15.325, -83.632, 50.734]
  MoveL 4639 to (498.02, 492.08, 10.1) mm, rotated rx 0 ry 90 rz 0 deg; joints [-11.318, -27.42, 111.703, -15.312, -83.622, 50.736]
  Set speed (120.0 mm/s)
  MoveL 4640 to (500.75, 492.32, 10.1) mm, rotated rx 0 ry 90 rz 0 deg; joints [-11.29, -27.37, 111.371, -15.292, -83.349, 50.808]
  Set speed (1000.0 mm/s)
  MoveL 4641 to (501, 491.11, 10.1) mm, rotated rx 0 ry 90 rz 0 deg; joints [-11.173, -27.37, 111.37, -15.175, -83.345, 50.796]
  Set speed (30.0 mm/s)
  Call Extruder(0.267)
  MoveL 4642 to (507.49, 497.59, 10.1) mm, rotated rx 0 ry 90 rz 0 deg; joints [-11.646, -27.224, 110.436, -15.677, -82.599, 51.059]
  MoveL 4643 to (507.61, 497.71, 10.1) mm, rotated rx 0 ry 90 rz 0 deg; joints [-11.655, -27.221, 110.418, -15.686, -82.585, 51.064]
  Set speed (120.0 mm/s)
  MoveL 4644 to (509.32, 490.68, 10.1) mm, rotated rx 0 ry 90 rz 0 deg; joints [-10.985, -27.216, 110.382, -15.013, -82.535, 50.994]
  Set speed (30.0 mm/s)
  Call Extruder(0.767)
  MoveL 4645 to (490.68, 509.32, 10.1) mm, rotated rx 0 ry 90 rz 0 deg; joints [-13.056, -27.482, 112.131, -17.049, -84.021, 50.795]
  MoveL 4646 to (490.56, 509.44, 10.1) mm, rotated rx 0 ry 90 rz 0 deg; joints [-13.07, -27.484, 112.142, -17.062, -84.03, 50.793]
  Set speed (120.0 mm/s)
  MoveL 4647 to (500.8, 492.37, 10.1) mm, rotated rx 0 ry 90 rz 0 deg; joints [-11.293, -27.369, 111.365, -15.296, -83.344, 50.81]
  Set speed (1000.0 mm/s)
  MoveL 4648 to (500.73, 492.3, 10.1) mm, rotated rx 0 ry 90 rz 0 deg; joints [-11.288, -27.371, 111.375, -15.29, -83.352, 50.807]
  Set speed (15.0 mm/s)
  Call Extruder(0.055)
  MoveL 4649 to (500.73, 490.41, 10.1) mm, rotated rx 0 ry 90 rz 0 deg; joints [-11.114, -27.378, 111.419, -15.114, -83.384, 50.779]
  Call Extruder(0.101)
  MoveL 4650 to (504.2, 490.4, 10.1) mm, rotated rx 0 ry 90 rz 0 deg; joints [-11.051, -27.314, 111.003, -15.061, -83.042, 50.865]
  Call Extruder(0.157)
  MoveL 4651 to (509.6, 490.4, 10.1) mm, rotated rx 0 ry 90 rz 0 deg; joints [-10.955, -27.211, 110.355, -14.983, -82.512, 50.997]
  Call Extruder(0.217)
  MoveL 4652 to (509.6, 497.87, 10.1) mm, rotated rx 0 ry 90 rz 0 deg; joints [-11.632, -27.182, 110.175, -15.67, -82.389, 51.116]
  Call Extruder(0.056)
  MoveL 4653 to (507.66, 497.87, 10.1) mm, rotated rx 0 ry 90 rz 0 deg; joints [-11.668, -27.22, 110.408, -15.7, -82.577, 51.068]
  Call Extruder(0.100)
  MoveL 4654 to (507.66, 501.31, 10.1) mm, rotated rx 0 ry 90 rz 0 deg; joints [-11.98, -27.206, 110.321, -16.017, -82.518, 51.124]
  Call Extruder(0.056)
  MoveL 4655 to (509.6, 501.32, 10.1) mm, rotated rx 0 ry 90 rz 0 deg; joints [-11.943, -27.168, 110.088, -15.987, -82.329, 51.173]
  Call Extruder(0.241)
  MoveL 4656 to (509.6, 509.6, 10.1) mm, rotated rx 0 ry 90 rz 0 deg; joints [-12.688, -27.132, 109.87, -16.745, -82.181, 51.315]
  Call Extruder(0.559)
  MoveL 4657 to (490.4, 509.6, 10.1) mm, rotated rx 0 ry 90 rz 0 deg; joints [-13.088, -27.486, 112.156, -17.08, -84.042, 50.791]
  MoveL 4658 to (490.4, 490.4, 10.1) mm, rotated rx 0 ry 90 rz 0 deg; joints [-11.303, -27.554, 112.646, -15.275, -84.402, 50.52]
  Call Extruder(0.226)
  MoveL 4659 to (498.18, 490.4, 10.1) mm, rotated rx 0 ry 90 rz 0 deg; joints [-11.159, -27.423, 111.724, -15.152, -83.635, 50.716]
  Call Extruder(0.055)
  MoveL 4660 to (498.18, 492.29, 10.1) mm, rotated rx 0 ry 90 rz 0 deg; joints [-11.334, -27.416, 111.679, -15.329, -83.603, 50.743]
  Call Extruder(0.029)
  MoveL 4661 to (499.18, 492.3, 10.1) mm, rotated rx 0 ry 90 rz 0 deg; joints [-11.316, -27.399, 111.559, -15.314, -83.504, 50.768]
  Call Extruder(0.045)
  MoveL 4662 to (500.73, 492.3, 10.1) mm, rotated rx 0 ry 90 rz 0 deg; joints [-11.288, -27.371, 111.375, -15.29, -83.352, 50.807]
  Set speed (120.0 mm/s)
  MoveL 4663 to (500.73, 491.9, 10.1) mm, rotated rx 0 ry 90 rz 0 deg; joints [-11.251, -27.372, 111.384, -15.253, -83.359, 50.801]
  Set speed (1000.0 mm/s)
  MoveL 4664 to (501.43, 491.9, 10.1) mm, rotated rx 0 ry 90 rz 0 deg; joints [-11.238, -27.36, 111.301, -15.242, -83.29, 50.818]
  Set speed (1000.0 mm/s)
  MoveL 4665 to (498.15, 492.32, 10.1) mm, rotated rx 0 ry 90 rz 0 deg; joints [-11.337, -27.417, 111.682, -15.332, -83.605, 50.742]
  Set speed (1000.0 mm/s)
  MoveL 4666 to (490.68, 490.68, 10.1) mm, rotated rx 0 ry 90 rz 0 deg; joints [-11.324, -27.549, 112.606, -15.297, -84.37, 50.531]
  Set speed (1000.0 mm/s)
  MoveL 4667 to (490.68, 490.68, 10.2) mm, rotated rx 0 ry 90 rz 0 deg; joints [-11.324, -27.56, 112.612, -15.297, -84.364, 50.532]
  Set speed (30.0 mm/s)
  Call Extruder(0.767)
  MoveL 4668 to (509.32, 509.32, 10.2) mm, rotated rx 0 ry 90 rz 0 deg; joints [-12.669, -27.149, 109.917, -16.725, -82.208, 51.304]
  MoveL 4669 to (509.44, 509.44, 10.2) mm, rotated rx 0 ry 90 rz 0 deg; joints [-12.677, -27.146, 109.899, -16.734, -82.194, 51.31]
  Set speed (120.0 mm/s)
  MoveL 4670 to (508.25, 501.65, 10.2) mm, rotated rx 0 ry 90 rz 0 deg; joints [-11.999, -27.203, 110.248, -16.039, -82.45, 51.146]
  Set speed (30.0 mm/s)
  Call Extruder(0.316)
  MoveL 4671 to (500.58, 509.32, 10.2) mm, rotated rx 0 ry 90 rz 0 deg; joints [-12.847, -27.318, 110.963, -16.872, -83.055, 51.069]
  Set speed (120.0 mm/s)
  MoveL 4672 to (499.42, 509.32, 10.2) mm, rotated rx 0 ry 90 rz 0 deg; joints [-12.872, -27.339, 111.101, -16.892, -83.167, 51.037]
  Set speed (30.0 mm/s)
  Call Extruder(0.360)
  MoveL 4673 to (490.68, 500.58, 10.2) mm, rotated rx 0 ry 90 rz 0 deg; joints [-12.247, -27.526, 112.368, -16.23, -84.184, 50.668]
  Set speed (120.0 mm/s)
  MoveL 4674 to (490.68, 499.42, 10.2) mm, rotated rx 0 ry 90 rz 0 deg; joints [-12.139, -27.53, 112.397, -16.121, -84.206, 50.651]
  Set speed (30.0 mm/s)
  Call Extruder(0.295)
  MoveL 4675 to (497.86, 492.24, 10.2) mm, rotated rx 0 ry 90 rz 0 deg; joints [-11.336, -27.433, 111.723, -15.33, -83.63, 50.735]
  MoveL 4676 to (497.98, 492.12, 10.2) mm, rotated rx 0 ry 90 rz 0 deg; joints [-11.322, -27.431, 111.712, -15.316, -83.62, 50.737]
  Set speed (120.0 mm/s)
  MoveL 4677 to (500.82, 492.32, 10.2) mm, rotated rx 0 ry 90 rz 0 deg; joints [-11.288, -27.38, 111.368, -15.291, -83.338, 50.811]
  Set speed (1000.0 mm/s)
  MoveL 4678 to (501.07, 491.17, 10.2) mm, rotated rx 0 ry 90 rz 0 deg; joints [-11.178, -27.379, 111.366, -15.18, -83.332, 50.8]
  Set speed (30.0 mm/s)
  Call Extruder(0.262)
  MoveL 4679 to (507.43, 497.53, 10.2) mm, rotated rx 0 ry 90 rz 0 deg; joints [-11.642, -27.236, 110.45, -15.673, -82.601, 51.058]
  MoveL 4680 to (507.55, 497.65, 10.2) mm, rotated rx 0 ry 90 rz 0 deg; joints [-11.65, -27.233, 110.432, -15.682, -82.587, 51.063]
  Set speed (120.0 mm/s)
  MoveL 4681 to (509.32, 490.68, 10.2) mm, rotated rx 0 ry 90 rz 0 deg; joints [-10.985, -27.226, 110.387, -15.013, -82.53, 50.996]
  Set speed (30.0 mm/s)
  Call Extruder(0.767)
  MoveL 4682 to (490.68, 509.32, 10.2) mm, rotated rx 0 ry 90 rz 0 deg; joints [-13.056, -27.493, 112.136, -17.049, -84.015, 50.797]
  MoveL 4683 to (490.56, 509.44, 10.2) mm, rotated rx 0 ry 90 rz 0 deg; joints [-13.07, -27.494, 112.148, -17.063, -84.025, 50.795]
  Set speed (120.0 mm/s)
  MoveL 4684 to (498.07, 492.37, 10.2) mm, rotated rx 0 ry 90 rz 0 deg; joints [-11.343, -27.429, 111.695, -15.338, -83.607, 50.742]
  Set speed (1000.0 mm/s)
  MoveL 4685 to (498.14, 492.3, 10.2) mm, rotated rx 0 ry 90 rz 0 deg; joints [-11.336, -27.428, 111.689, -15.331, -83.601, 50.743]
  Set speed (15.0 mm/s)
  Call Extruder(0.010)
  MoveL 4686 to (498.49, 492.3, 10.2) mm, rotated rx 0 ry 90 rz 0 deg; joints [-11.329, -27.421, 111.647, -15.325, -83.567, 50.752]
  Call Extruder(0.067)
  MoveL 4687 to (500.79, 492.3, 10.2) mm, rotated rx 0 ry 90 rz 0 deg; joints [-11.286, -27.38, 111.372, -15.289, -83.341, 50.81]
  Call Extruder(0.055)
  MoveL 4688 to (500.79, 490.4, 10.2) mm, rotated rx 0 ry 90 rz 0 deg; joints [-11.112, -27.387, 111.417, -15.113, -83.373, 50.782]
  Call Extruder(0.256)
  MoveL 4689 to (509.6, 490.4, 10.2) mm, rotated rx 0 ry 90 rz 0 deg; joints [-10.955, -27.222, 110.36, -14.983, -82.507, 50.998]
  Call Extruder(0.216)
  MoveL 4690 to (509.6, 497.81, 10.2) mm, rotated rx 0 ry 90 rz 0 deg; joints [-11.626, -27.193, 110.182, -15.665, -82.384, 51.117]
  Call Extruder(0.056)
  MoveL 4691 to (507.66, 497.81, 10.2) mm, rotated rx 0 ry 90 rz 0 deg; joints [-11.663, -27.23, 110.414, -15.695, -82.573, 51.068]
  Call Extruder(0.104)
  MoveL 4692 to (507.66, 501.37, 10.2) mm, rotated rx 0 ry 90 rz 0 deg; joints [-11.985, -27.216, 110.325, -16.022, -82.512, 51.126]
  Call Extruder(0.056)
  MoveL 4693 to (509.6, 501.37, 10.2) mm, rotated rx 0 ry 90 rz 0 deg; joints [-11.948, -27.178, 110.092, -15.992, -82.323, 51.176]
  Call Extruder(0.239)
  MoveL 4694 to (509.6, 509.6, 10.2) mm, rotated rx 0 ry 90 rz 0 deg; joints [-12.688, -27.142, 109.876, -16.746, -82.176, 51.317]
  Call Extruder(0.559)
  MoveL 4695 to (490.4, 509.6, 10.2) mm, rotated rx 0 ry 90 rz 0 deg; joints [-13.088, -27.496, 112.162, -17.08, -84.037, 50.793]
  MoveL 4696 to (490.4, 490.4, 10.2) mm, rotated rx 0 ry 90 rz 0 deg; joints [-11.303, -27.565, 112.651, -15.275, -84.397, 50.521]
  Call Extruder(0.225)
  MoveL 4697 to (498.14, 490.4, 10.2) mm, rotated rx 0 ry 90 rz 0 deg; joints [-11.16, -27.434, 111.733, -15.153, -83.634, 50.716]
  Call Extruder(0.045)
  MoveL 4698 to (498.14, 491.95, 10.2) mm, rotated rx 0 ry 90 rz 0 deg; joints [-11.303, -27.429, 111.697, -15.298, -83.607, 50.738]
  Call Extruder(0.007)
  MoveL 4699 to (498.14, 492.3, 10.2) mm, rotated rx 0 ry 90 rz 0 deg; joints [-11.336, -27.428, 111.689, -15.331, -83.601, 50.743]
  Set speed (120.0 mm/s)
  MoveL 4700 to (498.49, 492.3, 10.2) mm, rotated rx 0 ry 90 rz 0 deg; joints [-11.329, -27.421, 111.647, -15.325, -83.567, 50.752]
  Set speed (1000.0 mm/s)
  MoveL 4701 to (498.54, 492.3, 10.2) mm, rotated rx 0 ry 90 rz 0 deg; joints [-11.328, -27.421, 111.641, -15.324, -83.562, 50.753]
  Set speed (1000.0 mm/s)
  MoveL 4702 to (498.54, 493, 10.2) mm, rotated rx 0 ry 90 rz 0 deg; joints [-11.393, -27.418, 111.624, -15.39, -83.55, 50.763]
  Set speed (1000.0 mm/s)
  MoveL 4703 to (490.68, 490.68, 10.2) mm, rotated rx 0 ry 90 rz 0 deg; joints [-11.324, -27.56, 112.612, -15.297, -84.364, 50.532]
  Set speed (1000.0 mm/s)
  MoveL 4704 to (490.68, 490.68, 10.3) mm, rotated rx 0 ry 90 rz 0 deg; joints [-11.324, -27.57, 112.617, -15.297, -84.359, 50.533]
  Set speed (30.0 mm/s)
  Call Extruder(0.767)
  MoveL 4705 to (509.32, 509.32, 10.3) mm, rotated rx 0 ry 90 rz 0 deg; joints [-12.669, -27.159, 109.922, -16.725, -82.203, 51.306]
  MoveL 4706 to (509.44, 509.44, 10.3) mm, rotated rx 0 ry 90 rz 0 deg; joints [-12.677, -27.156, 109.904, -16.734, -82.189, 51.311]
  Set speed (120.0 mm/s)
  MoveL 4707 to (508.19, 501.71, 10.3) mm, rotated rx 0 ry 90 rz 0 deg; joints [-12.005, -27.215, 110.258, -16.045, -82.449, 51.147]
  Set speed (30.0 mm/s)
  Call Extruder(0.313)
  MoveL 4708 to (500.58, 509.32, 10.3) mm, rotated rx 0 ry 90 rz 0 deg; joints [-12.847, -27.328, 110.969, -16.872, -83.05, 51.07]
  Set speed (120.0 mm/s)
  MoveL 4709 to (499.42, 509.32, 10.3) mm, rotated rx 0 ry 90 rz 0 deg; joints [-12.872, -27.349, 111.107, -16.892, -83.162, 51.039]
  Set speed (30.0 mm/s)
  Call Extruder(0.360)
  MoveL 4710 to (490.68, 500.58, 10.3) mm, rotated rx 0 ry 90 rz 0 deg; joints [-12.247, -27.536, 112.373, -16.23, -84.179, 50.669]
  Set speed (120.0 mm/s)
  MoveL 4711 to (490.68, 499.42, 10.3) mm, rotated rx 0 ry 90 rz 0 deg; joints [-12.139, -27.54, 112.403, -16.121, -84.201, 50.653]
  Set speed (30.0 mm/s)
  Call Extruder(0.293)
  MoveL 4712 to (497.8, 492.3, 10.3) mm, rotated rx 0 ry 90 rz 0 deg; joints [-11.342, -27.444, 111.734, -15.336, -83.629, 50.736]
  MoveL 4713 to (497.92, 492.17, 10.3) mm, rotated rx 0 ry 90 rz 0 deg; joints [-11.328, -27.442, 111.722, -15.322, -83.619, 50.737]
  Set speed (120.0 mm/s)
  MoveL 4714 to (500.88, 492.32, 10.3) mm, rotated rx 0 ry 90 rz 0 deg; joints [-11.287, -27.389, 111.366, -15.291, -83.326, 50.814]
  Set speed (1000.0 mm/s)
  MoveL 4715 to (501.13, 491.23, 10.3) mm, rotated rx 0 ry 90 rz 0 deg; joints [-11.183, -27.389, 111.362, -15.185, -83.32, 50.804]
  Set speed (30.0 mm/s)
  Call Extruder(0.257)
  MoveL 4716 to (507.38, 497.48, 10.3) mm, rotated rx 0 ry 90 rz 0 deg; joints [-11.638, -27.248, 110.461, -15.669, -82.601, 51.057]
  MoveL 4717 to (507.51, 497.61, 10.3) mm, rotated rx 0 ry 90 rz 0 deg; joints [-11.647, -27.245, 110.444, -15.679, -82.587, 51.062]
  Set speed (120.0 mm/s)
  MoveL 4718 to (509.32, 490.68, 10.3) mm, rotated rx 0 ry 90 rz 0 deg; joints [-10.985, -27.237, 110.392, -15.013, -82.525, 50.997]
  Set speed (30.0 mm/s)
  Call Extruder(0.767)
  MoveL 4719 to (490.68, 509.32, 10.3) mm, rotated rx 0 ry 90 rz 0 deg; joints [-13.056, -27.503, 112.142, -17.049, -84.01, 50.798]
  MoveL 4720 to (490.56, 509.44, 10.3) mm, rotated rx 0 ry 90 rz 0 deg; joints [-13.07, -27.505, 112.153, -17.063, -84.02, 50.797]
  Set speed (120.0 mm/s)
  MoveL 4721 to (498.01, 492.37, 10.3) mm, rotated rx 0 ry 90 rz 0 deg; joints [-11.344, -27.44, 111.707, -15.339, -83.607, 50.742]
  Set speed (1000.0 mm/s)
  MoveL 4722 to (498.08, 492.3, 10.3) mm, rotated rx 0 ry 90 rz 0 deg; joints [-11.337, -27.439, 111.7, -15.332, -83.602, 50.743]
  Set speed (15.0 mm/s)
  Call Extruder(0.010)
  MoveL 4723 to (498.43, 492.3, 10.3) mm, rotated rx 0 ry 90 rz 0 deg; joints [-11.33, -27.433, 111.659, -15.326, -83.567, 50.752]
  Call Extruder(0.070)
  MoveL 4724 to (500.85, 492.3, 10.3) mm, rotated rx 0 ry 90 rz 0 deg; joints [-11.285, -27.39, 111.37, -15.288, -83.329, 50.813]
  Call Extruder(0.055)
  MoveL 4725 to (500.85, 490.4, 10.3) mm, rotated rx 0 ry 90 rz 0 deg; joints [-11.111, -27.397, 111.415, -15.112, -83.361, 50.785]
  Call Extruder(0.255)
  MoveL 4726 to (509.6, 490.4, 10.3) mm, rotated rx 0 ry 90 rz 0 deg; joints [-10.955, -27.232, 110.365, -14.983, -82.502, 51]
  Call Extruder(0.214)
  MoveL 4727 to (509.6, 497.75, 10.3) mm, rotated rx 0 ry 90 rz 0 deg; joints [-11.621, -27.203, 110.188, -15.66, -82.38, 51.117]
  Call Extruder(0.056)
  MoveL 4728 to (507.66, 497.75, 10.3) mm, rotated rx 0 ry 90 rz 0 deg; joints [-11.657, -27.241, 110.421, -15.689, -82.569, 51.069]
  Call Extruder(0.107)
  MoveL 4729 to (507.66, 501.43, 10.3) mm, rotated rx 0 ry 90 rz 0 deg; joints [-11.99, -27.226, 110.329, -16.028, -82.506, 51.128]
  Call Extruder(0.056)
  MoveL 4730 to (509.6, 501.43, 10.3) mm, rotated rx 0 ry 90 rz 0 deg; joints [-11.953, -27.188, 110.096, -15.998, -82.317, 51.178]
  Call Extruder(0.238)
  MoveL 4731 to (509.6, 509.6, 10.3) mm, rotated rx 0 ry 90 rz 0 deg; joints [-12.688, -27.152, 109.881, -16.746, -82.171, 51.318]
  Call Extruder(0.559)
  MoveL 4732 to (490.4, 509.6, 10.3) mm, rotated rx 0 ry 90 rz 0 deg; joints [-13.088, -27.507, 112.167, -17.08, -84.032, 50.795]
  MoveL 4733 to (490.4, 490.4, 10.3) mm, rotated rx 0 ry 90 rz 0 deg; joints [-11.303, -27.576, 112.657, -15.275, -84.392, 50.523]
  Call Extruder(0.224)
  MoveL 4734 to (498.08, 490.4, 10.3) mm, rotated rx 0 ry 90 rz 0 deg; joints [-11.161, -27.446, 111.745, -15.154, -83.634, 50.716]
  Call Extruder(0.045)
  MoveL 4735 to (498.08, 491.95, 10.3) mm, rotated rx 0 ry 90 rz 0 deg; joints [-11.304, -27.44, 111.709, -15.299, -83.608, 50.738]
  Call Extruder(0.007)
  MoveL 4736 to (498.08, 492.3, 10.3) mm, rotated rx 0 ry 90 rz 0 deg; joints [-11.337, -27.439, 111.7, -15.332, -83.602, 50.743]
  Set speed (120.0 mm/s)
  MoveL 4737 to (498.43, 492.3, 10.3) mm, rotated rx 0 ry 90 rz 0 deg; joints [-11.33, -27.433, 111.659, -15.326, -83.567, 50.752]
  Set speed (1000.0 mm/s)
  MoveL 4738 to (498.48, 492.3, 10.3) mm, rotated rx 0 ry 90 rz 0 deg; joints [-11.329, -27.432, 111.653, -15.325, -83.562, 50.753]
  Set speed (1000.0 mm/s)
  MoveL 4739 to (498.48, 493, 10.3) mm, rotated rx 0 ry 90 rz 0 deg; joints [-11.394, -27.43, 111.636, -15.391, -83.55, 50.763]
  Set speed (1000.0 mm/s)
  MoveL 4740 to (490.68, 490.68, 10.3) mm, rotated rx 0 ry 90 rz 0 deg; joints [-11.324, -27.57, 112.617, -15.297, -84.359, 50.533]
  Set speed (1000.0 mm/s)
  MoveL 4741 to (490.68, 490.68, 10.4) mm, rotated rx 0 ry 90 rz 0 deg; joints [-11.324, -27.581, 112.622, -15.297, -84.354, 50.535]
  Set speed (30.0 mm/s)
  Call Extruder(0.767)
  MoveL 4742 to (509.32, 509.32, 10.4) mm, rotated rx 0 ry 90 rz 0 deg; joints [-12.669, -27.17, 109.927, -16.725, -82.198, 51.307]
  MoveL 4743 to (509.44, 509.44, 10.4) mm, rotated rx 0 ry 90 rz 0 deg; joints [-12.677, -27.167, 109.909, -16.734, -82.184, 51.313]
  Set speed (120.0 mm/s)
  MoveL 4744 to (508.14, 501.76, 10.4) mm, rotated rx 0 ry 90 rz 0 deg; joints [-12.011, -27.226, 110.269, -16.051, -82.449, 51.148]
  Set speed (30.0 mm/s)
  Call Extruder(0.311)
  MoveL 4745 to (500.58, 509.32, 10.4) mm, rotated rx 0 ry 90 rz 0 deg; joints [-12.847, -27.339, 110.974, -16.872, -83.045, 51.072]
  Set speed (120.0 mm/s)
  MoveL 4746 to (499.42, 509.32, 10.4) mm, rotated rx 0 ry 90 rz 0 deg; joints [-12.872, -27.36, 111.112, -16.892, -83.157, 51.04]
  Set speed (30.0 mm/s)
  Call Extruder(0.360)
  MoveL 4747 to (490.68, 500.58, 10.4) mm, rotated rx 0 ry 90 rz 0 deg; joints [-12.247, -27.547, 112.378, -16.23, -84.174, 50.671]
  Set speed (120.0 mm/s)
  MoveL 4748 to (490.68, 499.42, 10.4) mm, rotated rx 0 ry 90 rz 0 deg; joints [-12.139, -27.551, 112.408, -16.121, -84.196, 50.654]
  Set speed (30.0 mm/s)
  Call Extruder(0.291)
  MoveL 4749 to (497.74, 492.35, 10.4) mm, rotated rx 0 ry 90 rz 0 deg; joints [-11.348, -27.456, 111.745, -15.342, -83.629, 50.737]
  MoveL 4750 to (497.87, 492.23, 10.4) mm, rotated rx 0 ry 90 rz 0 deg; joints [-11.334, -27.454, 111.733, -15.329, -83.619, 50.738]
  Set speed (120.0 mm/s)
  MoveL 4751 to (500.95, 492.32, 10.4) mm, rotated rx 0 ry 90 rz 0 deg; joints [-11.286, -27.399, 111.363, -15.29, -83.315, 50.817]
  Set speed (1000.0 mm/s)
  MoveL 4752 to (501.2, 491.3, 10.4) mm, rotated rx 0 ry 90 rz 0 deg; joints [-11.187, -27.398, 111.358, -15.19, -83.307, 50.808]
  Set speed (30.0 mm/s)
  Call Extruder(0.255)
  MoveL 4753 to (507.39, 497.49, 10.4) mm, rotated rx 0 ry 90 rz 0 deg; joints [-11.638, -27.258, 110.466, -15.669, -82.596, 51.059]
  MoveL 4754 to (507.51, 497.61, 10.4) mm, rotated rx 0 ry 90 rz 0 deg; joints [-11.647, -27.255, 110.449, -15.679, -82.582, 51.064]
  Set speed (120.0 mm/s)
  MoveL 4755 to (509.32, 490.68, 10.4) mm, rotated rx 0 ry 90 rz 0 deg; joints [-10.985, -27.247, 110.398, -15.013, -82.52, 50.999]
  Set speed (30.0 mm/s)
  Call Extruder(0.767)
  MoveL 4756 to (490.68, 509.32, 10.4) mm, rotated rx 0 ry 90 rz 0 deg; joints [-13.056, -27.514, 112.147, -17.049, -84.005, 50.8]
  MoveL 4757 to (490.56, 509.44, 10.4) mm, rotated rx 0 ry 90 rz 0 deg; joints [-13.07, -27.516, 112.158, -17.063, -84.015, 50.798]
  Set speed (120.0 mm/s)
  MoveL 4758 to (497.96, 492.37, 10.4) mm, rotated rx 0 ry 90 rz 0 deg; joints [-11.345, -27.452, 111.719, -15.34, -83.608, 50.742]
  Set speed (1000.0 mm/s)
  MoveL 4759 to (498.03, 492.3, 10.4) mm, rotated rx 0 ry 90 rz 0 deg; joints [-11.338, -27.451, 111.712, -15.333, -83.602, 50.743]
  Set speed (15.0 mm/s)
  Call Extruder(0.010)
  MoveL 4760 to (498.37, 492.3, 10.4) mm, rotated rx 0 ry 90 rz 0 deg; joints [-11.331, -27.445, 111.671, -15.327, -83.568, 50.752]
  Call Extruder(0.074)
  MoveL 4761 to (500.92, 492.3, 10.4) mm, rotated rx 0 ry 90 rz 0 deg; joints [-11.284, -27.399, 111.367, -15.288, -83.318, 50.816]
  Call Extruder(0.055)
  MoveL 4762 to (500.92, 490.4, 10.4) mm, rotated rx 0 ry 90 rz 0 deg; joints [-11.11, -27.406, 111.412, -15.111, -83.35, 50.788]
  Call Extruder(0.253)
  MoveL 4763 to (509.6, 490.4, 10.4) mm, rotated rx 0 ry 90 rz 0 deg; joints [-10.955, -27.243, 110.37, -14.983, -82.497, 51.001]
  Call Extruder(0.212)
  MoveL 4764 to (509.6, 497.69, 10.4) mm, rotated rx 0 ry 90 rz 0 deg; joints [-11.615, -27.214, 110.195, -15.655, -82.376, 51.118]
  Call Extruder(0.056)
  MoveL 4765 to (507.67, 497.69, 10.4) mm, rotated rx 0 ry 90 rz 0 deg; joints [-11.652, -27.252, 110.428, -15.684, -82.565, 51.069]
  Call Extruder(0.110)
  MoveL 4766 to (507.66, 501.48, 10.4) mm, rotated rx 0 ry 90 rz 0 deg; joints [-11.995, -27.237, 110.333, -16.033, -82.5, 51.131]
  Call Extruder(0.056)
  MoveL 4767 to (509.6, 501.49, 10.4) mm, rotated rx 0 ry 90 rz 0 deg; joints [-11.958, -27.198, 110.099, -16.003, -82.311, 51.181]
  Call Extruder(0.236)
  MoveL 4768 to (509.6, 509.6, 10.4) mm, rotated rx 0 ry 90 rz 0 deg; joints [-12.688, -27.163, 109.886, -16.746, -82.166, 51.32]
  Call Extruder(0.559)
  MoveL 4769 to (490.4, 509.6, 10.4) mm, rotated rx 0 ry 90 rz 0 deg; joints [-13.088, -27.518, 112.172, -17.081, -84.027, 50.796]
  MoveL 4770 to (490.4, 490.4, 10.4) mm, rotated rx 0 ry 90 rz 0 deg; joints [-11.303, -27.586, 112.662, -15.275, -84.386, 50.524]
  Call Extruder(0.212)
  MoveL 4771 to (497.68, 490.4, 10.4) mm, rotated rx 0 ry 90 rz 0 deg; joints [-11.169, -27.464, 111.799, -15.16, -83.669, 50.707]
  Call Extruder(0.010)
  MoveL 4772 to (498.03, 490.4, 10.4) mm, rotated rx 0 ry 90 rz 0 deg; joints [-11.162, -27.457, 111.757, -15.155, -83.635, 50.716]
  Call Extruder(0.007)
  MoveL 4773 to (498.03, 490.75, 10.4) mm, rotated rx 0 ry 90 rz 0 deg; joints [-11.195, -27.456, 111.749, -15.188, -83.629, 50.721]
  Call Extruder(0.035)
  MoveL 4774 to (498.03, 491.95, 10.4) mm, rotated rx 0 ry 90 rz 0 deg; joints [-11.305, -27.452, 111.721, -15.3, -83.608, 50.738]
  Call Extruder(0.007)
  MoveL 4775 to (498.03, 492.3, 10.4) mm, rotated rx 0 ry 90 rz 0 deg; joints [-11.338, -27.451, 111.712, -15.333, -83.602, 50.743]
  Set speed (120.0 mm/s)
  MoveL 4776 to (498.37, 492.3, 10.4) mm, rotated rx 0 ry 90 rz 0 deg; joints [-11.331, -27.445, 111.671, -15.327, -83.568, 50.752]
  Set speed (1000.0 mm/s)
  MoveL 4777 to (498.43, 492.3, 10.4) mm, rotated rx 0 ry 90 rz 0 deg; joints [-11.33, -27.444, 111.665, -15.326, -83.563, 50.753]
  Set speed (1000.0 mm/s)
  MoveL 4778 to (498.42, 493, 10.4) mm, rotated rx 0 ry 90 rz 0 deg; joints [-11.395, -27.441, 111.648, -15.392, -83.551, 50.763]
  Set speed (1000.0 mm/s)
  MoveL 4779 to (490.68, 490.68, 10.4) mm, rotated rx 0 ry 90 rz 0 deg; joints [-11.324, -27.581, 112.622, -15.297, -84.354, 50.535]
  Set speed (1000.0 mm/s)
  MoveL 4780 to (490.68, 490.68, 10.5) mm, rotated rx 0 ry 90 rz 0 deg; joints [-11.324, -27.592, 112.627, -15.297, -84.349, 50.536]
  Set speed (30.0 mm/s)
  Call Extruder(0.767)
  MoveL 4781 to (509.32, 509.32, 10.5) mm, rotated rx 0 ry 90 rz 0 deg; joints [-12.669, -27.18, 109.933, -16.725, -82.193, 51.309]
  MoveL 4782 to (509.44, 509.44, 10.5) mm, rotated rx 0 ry 90 rz 0 deg; joints [-12.677, -27.177, 109.914, -16.734, -82.179, 51.314]
  Set speed (120.0 mm/s)
  MoveL 4783 to (508.08, 501.82, 10.5) mm, rotated rx 0 ry 90 rz 0 deg; joints [-12.018, -27.237, 110.279, -16.058, -82.448, 51.149]
  Set speed (30.0 mm/s)
  Call Extruder(0.309)
  MoveL 4784 to (500.58, 509.32, 10.5) mm, rotated rx 0 ry 90 rz 0 deg; joints [-12.847, -27.349, 110.979, -16.873, -83.04, 51.074]
  Set speed (120.0 mm/s)
  MoveL 4785 to (499.42, 509.32, 10.5) mm, rotated rx 0 ry 90 rz 0 deg; joints [-12.872, -27.371, 111.117, -16.893, -83.152, 51.042]
  Set speed (30.0 mm/s)
  Call Extruder(0.360)
  MoveL 4786 to (490.68, 500.58, 10.5) mm, rotated rx 0 ry 90 rz 0 deg; joints [-12.247, -27.558, 112.384, -16.23, -84.169, 50.672]
  Set speed (120.0 mm/s)
  MoveL 4787 to (490.68, 499.42, 10.5) mm, rotated rx 0 ry 90 rz 0 deg; joints [-12.139, -27.562, 112.413, -16.121, -84.191, 50.656]
  Set speed (30.0 mm/s)
  Call Extruder(0.288)
  MoveL 4788 to (497.69, 492.41, 10.5) mm, rotated rx 0 ry 90 rz 0 deg; joints [-11.354, -27.467, 111.755, -15.349, -83.628, 50.738]
  MoveL 4789 to (497.81, 492.29, 10.5) mm, rotated rx 0 ry 90 rz 0 deg; joints [-11.341, -27.465, 111.743, -15.335, -83.618, 50.739]
  Set speed (120.0 mm/s)
  MoveL 4790 to (501.01, 492.33, 10.5) mm, rotated rx 0 ry 90 rz 0 deg; joints [-11.285, -27.408, 111.361, -15.289, -83.303, 50.82]
  Set speed (1000.0 mm/s)
  MoveL 4791 to (501.26, 491.36, 10.5) mm, rotated rx 0 ry 90 rz 0 deg; joints [-11.192, -27.407, 111.354, -15.196, -83.295, 50.812]
  Set speed (30.0 mm/s)
  Call Extruder(0.252)
  MoveL 4792 to (507.38, 497.48, 10.5) mm, rotated rx 0 ry 90 rz 0 deg; joints [-11.638, -27.269, 110.472, -15.67, -82.591, 51.06]
  MoveL 4793 to (507.51, 497.61, 10.5) mm, rotated rx 0 ry 90 rz 0 deg; joints [-11.647, -27.266, 110.454, -15.679, -82.577, 51.065]
  Set speed (120.0 mm/s)
  MoveL 4794 to (509.32, 490.68, 10.5) mm, rotated rx 0 ry 90 rz 0 deg; joints [-10.985, -27.258, 110.403, -15.013, -82.515, 51]
  Set speed (30.0 mm/s)
  Call Extruder(0.767)
  MoveL 4795 to (490.68, 509.32, 10.5) mm, rotated rx 0 ry 90 rz 0 deg; joints [-13.056, -27.525, 112.152, -17.049, -84, 50.801]
  MoveL 4796 to (490.56, 509.44, 10.5) mm, rotated rx 0 ry 90 rz 0 deg; joints [-13.07, -27.526, 112.163, -17.063, -84.009, 50.8]
  Set speed (120.0 mm/s)
  MoveL 4797 to (497.9, 492.37, 10.5) mm, rotated rx 0 ry 90 rz 0 deg; joints [-11.346, -27.463, 111.731, -15.341, -83.608, 50.742]
  Set speed (1000.0 mm/s)
  MoveL 4798 to (497.97, 492.3, 10.5) mm, rotated rx 0 ry 90 rz 0 deg; joints [-11.339, -27.462, 111.724, -15.334, -83.603, 50.743]
  Set speed (15.0 mm/s)
  Call Extruder(0.010)
  MoveL 4799 to (498.32, 492.3, 10.5) mm, rotated rx 0 ry 90 rz 0 deg; joints [-11.332, -27.456, 111.683, -15.328, -83.568, 50.752]
  Call Extruder(0.077)
  MoveL 4800 to (500.98, 492.3, 10.5) mm, rotated rx 0 ry 90 rz 0 deg; joints [-11.283, -27.409, 111.365, -15.287, -83.306, 50.819]
  Call Extruder(0.055)
  MoveL 4801 to (500.98, 490.4, 10.5) mm, rotated rx 0 ry 90 rz 0 deg; joints [-11.109, -27.415, 111.41, -15.11, -83.338, 50.791]
  Call Extruder(0.251)
  MoveL 4802 to (509.6, 490.4, 10.5) mm, rotated rx 0 ry 90 rz 0 deg; joints [-10.955, -27.253, 110.375, -14.984, -82.492, 51.002]
  Call Extruder(0.210)
  MoveL 4803 to (509.6, 497.63, 10.5) mm, rotated rx 0 ry 90 rz 0 deg; joints [-11.61, -27.225, 110.202, -15.649, -82.372, 51.118]
  Call Extruder(0.056)
  MoveL 4804 to (507.67, 497.63, 10.5) mm, rotated rx 0 ry 90 rz 0 deg; joints [-11.646, -27.263, 110.434, -15.679, -82.561, 51.069]
  Call Extruder(0.114)
  MoveL 4805 to (507.66, 501.54, 10.5) mm, rotated rx 0 ry 90 rz 0 deg; joints [-12, -27.247, 110.336, -16.039, -82.494, 51.133]
  Call Extruder(0.056)
  MoveL 4806 to (509.6, 501.54, 10.5) mm, rotated rx 0 ry 90 rz 0 deg; joints [-11.963, -27.209, 110.103, -16.009, -82.305, 51.183]
  Call Extruder(0.235)
  MoveL 4807 to (509.6, 509.6, 10.5) mm, rotated rx 0 ry 90 rz 0 deg; joints [-12.688, -27.173, 109.891, -16.746, -82.161, 51.321]
  Call Extruder(0.559)
  MoveL 4808 to (490.4, 509.6, 10.5) mm, rotated rx 0 ry 90 rz 0 deg; joints [-13.088, -27.528, 112.177, -17.081, -84.021, 50.798]
  MoveL 4809 to (490.4, 490.4, 10.5) mm, rotated rx 0 ry 90 rz 0 deg; joints [-11.303, -27.597, 112.667, -15.275, -84.381, 50.526]
  Call Extruder(0.210)
  MoveL 4810 to (497.62, 490.4, 10.5) mm, rotated rx 0 ry 90 rz 0 deg; joints [-11.17, -27.475, 111.811, -15.161, -83.669, 50.707]
  Call Extruder(0.010)
  MoveL 4811 to (497.97, 490.4, 10.5) mm, rotated rx 0 ry 90 rz 0 deg; joints [-11.163, -27.469, 111.769, -15.156, -83.635, 50.716]
  Call Extruder(0.007)
  MoveL 4812 to (497.97, 490.75, 10.5) mm, rotated rx 0 ry 90 rz 0 deg; joints [-11.196, -27.468, 111.761, -15.189, -83.629, 50.721]
  Call Extruder(0.035)
  MoveL 4813 to (497.97, 491.95, 10.5) mm, rotated rx 0 ry 90 rz 0 deg; joints [-11.306, -27.464, 111.733, -15.301, -83.609, 50.738]
  Call Extruder(0.007)
  MoveL 4814 to (497.97, 492.3, 10.5) mm, rotated rx 0 ry 90 rz 0 deg; joints [-11.339, -27.462, 111.724, -15.334, -83.603, 50.743]
  Set speed (120.0 mm/s)
  MoveL 4815 to (498.32, 492.3, 10.5) mm, rotated rx 0 ry 90 rz 0 deg; joints [-11.332, -27.456, 111.683, -15.328, -83.568, 50.752]
  Set speed (1000.0 mm/s)
  MoveL 4816 to (498.37, 492.3, 10.5) mm, rotated rx 0 ry 90 rz 0 deg; joints [-11.331, -27.455, 111.677, -15.327, -83.563, 50.753]
  Set speed (1000.0 mm/s)
  MoveL 4817 to (498.37, 493, 10.5) mm, rotated rx 0 ry 90 rz 0 deg; joints [-11.396, -27.453, 111.66, -15.393, -83.551, 50.763]
  Set speed (1000.0 mm/s)
  MoveL 4818 to (490.68, 490.68, 10.5) mm, rotated rx 0 ry 90 rz 0 deg; joints [-11.324, -27.592, 112.627, -15.297, -84.349, 50.536]
  Set speed (1000.0 mm/s)
  MoveL 4819 to (490.68, 490.68, 10.6) mm, rotated rx 0 ry 90 rz 0 deg; joints [-11.324, -27.602, 112.633, -15.297, -84.343, 50.538]
  Set speed (30.0 mm/s)
  Call Extruder(0.767)
  MoveL 4820 to (509.32, 509.32, 10.6) mm, rotated rx 0 ry 90 rz 0 deg; joints [-12.669, -27.191, 109.938, -16.725, -82.188, 51.31]
  MoveL 4821 to (509.44, 509.44, 10.6) mm, rotated rx 0 ry 90 rz 0 deg; joints [-12.677, -27.188, 109.92, -16.735, -82.174, 51.316]
  Set speed (120.0 mm/s)
  MoveL 4822 to (508.02, 501.88, 10.6) mm, rotated rx 0 ry 90 rz 0 deg; joints [-12.024, -27.249, 110.29, -16.064, -82.448, 51.149]
  Set speed (30.0 mm/s)
  Call Extruder(0.306)
  MoveL 4823 to (500.58, 509.32, 10.6) mm, rotated rx 0 ry 90 rz 0 deg; joints [-12.847, -27.36, 110.984, -16.873, -83.034, 51.075]
  Set speed (120.0 mm/s)
  MoveL 4824 to (499.42, 509.32, 10.6) mm, rotated rx 0 ry 90 rz 0 deg; joints [-12.872, -27.381, 111.122, -16.893, -83.147, 51.044]
  Set speed (30.0 mm/s)
  Call Extruder(0.360)
  MoveL 4825 to (490.68, 500.58, 10.6) mm, rotated rx 0 ry 90 rz 0 deg; joints [-12.247, -27.568, 112.389, -16.23, -84.164, 50.674]
  Set speed (120.0 mm/s)
  MoveL 4826 to (490.68, 499.42, 10.6) mm, rotated rx 0 ry 90 rz 0 deg; joints [-12.139, -27.572, 112.418, -16.121, -84.185, 50.658]
  Set speed (30.0 mm/s)
  Call Extruder(0.286)
  MoveL 4827 to (497.63, 492.47, 10.6) mm, rotated rx 0 ry 90 rz 0 deg; joints [-11.361, -27.478, 111.766, -15.355, -83.628, 50.739]
  MoveL 4828 to (497.76, 492.34, 10.6) mm, rotated rx 0 ry 90 rz 0 deg; joints [-11.347, -27.477, 111.754, -15.341, -83.618, 50.74]
  Set speed (120.0 mm/s)
  MoveL 4829 to (501.07, 492.32, 10.6) mm, rotated rx 0 ry 90 rz 0 deg; joints [-11.284, -27.417, 111.359, -15.288, -83.292, 50.823]
  Set speed (1000.0 mm/s)
  MoveL 4830 to (501.33, 491.43, 10.6) mm, rotated rx 0 ry 90 rz 0 deg; joints [-11.197, -27.416, 111.35, -15.201, -83.282, 50.816]
  Set speed (30.0 mm/s)
  Call Extruder(0.249)
  MoveL 4831 to (507.38, 497.48, 10.6) mm, rotated rx 0 ry 90 rz 0 deg; joints [-11.638, -27.279, 110.477, -15.67, -82.586, 51.061]
  MoveL 4832 to (507.51, 497.61, 10.6) mm, rotated rx 0 ry 90 rz 0 deg; joints [-11.647, -27.276, 110.459, -15.679, -82.572, 51.066]
  Set speed (120.0 mm/s)
  MoveL 4833 to (509.32, 490.68, 10.6) mm, rotated rx 0 ry 90 rz 0 deg; joints [-10.985, -27.268, 110.408, -15.014, -82.51, 51.001]
  Set speed (30.0 mm/s)
  Call Extruder(0.767)
  MoveL 4834 to (490.68, 509.32, 10.6) mm, rotated rx 0 ry 90 rz 0 deg; joints [-13.056, -27.535, 112.157, -17.049, -83.995, 50.803]
  MoveL 4835 to (490.56, 509.44, 10.6) mm, rotated rx 0 ry 90 rz 0 deg; joints [-13.07, -27.537, 112.169, -17.063, -84.004, 50.801]
  Set speed (120.0 mm/s)
  MoveL 4836 to (497.84, 492.37, 10.6) mm, rotated rx 0 ry 90 rz 0 deg; joints [-11.347, -27.475, 111.743, -15.342, -83.609, 50.742]
  Set speed (1000.0 mm/s)
  MoveL 4837 to (497.91, 492.3, 10.6) mm, rotated rx 0 ry 90 rz 0 deg; joints [-11.34, -27.474, 111.736, -15.335, -83.603, 50.743]
  Set speed (15.0 mm/s)
  Call Extruder(0.010)
  MoveL 4838 to (498.26, 492.3, 10.6) mm, rotated rx 0 ry 90 rz 0 deg; joints [-11.333, -27.468, 111.695, -15.329, -83.568, 50.752]
  Call Extruder(0.081)
  MoveL 4839 to (501.05, 492.3, 10.6) mm, rotated rx 0 ry 90 rz 0 deg; joints [-11.282, -27.418, 111.363, -15.286, -83.295, 50.822]
  Call Extruder(0.055)
  MoveL 4840 to (501.05, 490.4, 10.6) mm, rotated rx 0 ry 90 rz 0 deg; joints [-11.107, -27.425, 111.407, -15.109, -83.327, 50.794]
  Call Extruder(0.249)
  MoveL 4841 to (509.6, 490.4, 10.6) mm, rotated rx 0 ry 90 rz 0 deg; joints [-10.955, -27.264, 110.381, -14.984, -82.486, 51.004]
  Call Extruder(0.209)
  MoveL 4842 to (509.6, 497.57, 10.6) mm, rotated rx 0 ry 90 rz 0 deg; joints [-11.605, -27.235, 110.208, -15.644, -82.368, 51.119]
  Call Extruder(0.056)
  MoveL 4843 to (507.67, 497.57, 10.6) mm, rotated rx 0 ry 90 rz 0 deg; joints [-11.641, -27.273, 110.441, -15.673, -82.557, 51.07]
  Call Extruder(0.117)
  MoveL 4844 to (507.66, 501.6, 10.6) mm, rotated rx 0 ry 90 rz 0 deg; joints [-12.005, -27.257, 110.34, -16.044, -82.487, 51.136]
  Call Extruder(0.056)
  MoveL 4845 to (509.6, 501.6, 10.6) mm, rotated rx 0 ry 90 rz 0 deg; joints [-11.969, -27.219, 110.107, -16.014, -82.299, 51.186]
  Call Extruder(0.233)
  MoveL 4846 to (509.6, 509.6, 10.6) mm, rotated rx 0 ry 90 rz 0 deg; joints [-12.688, -27.184, 109.896, -16.747, -82.156, 51.323]
  Call Extruder(0.559)
  MoveL 4847 to (490.4, 509.6, 10.6) mm, rotated rx 0 ry 90 rz 0 deg; joints [-13.088, -27.539, 112.183, -17.081, -84.016, 50.799]
  MoveL 4848 to (490.4, 490.4, 10.6) mm, rotated rx 0 ry 90 rz 0 deg; joints [-11.303, -27.608, 112.672, -15.276, -84.376, 50.527]
  Call Extruder(0.219)
  MoveL 4849 to (497.91, 490.4, 10.6) mm, rotated rx 0 ry 90 rz 0 deg; joints [-11.164, -27.481, 111.781, -15.157, -83.635, 50.716]
  Call Extruder(0.045)
  MoveL 4850 to (497.91, 491.95, 10.6) mm, rotated rx 0 ry 90 rz 0 deg; joints [-11.307, -27.475, 111.745, -15.302, -83.609, 50.738]
  Call Extruder(0.007)
  MoveL 4851 to (497.91, 492.3, 10.6) mm, rotated rx 0 ry 90 rz 0 deg; joints [-11.34, -27.474, 111.736, -15.335, -83.603, 50.743]
  Set speed (120.0 mm/s)
  MoveL 4852 to (498.26, 492.3, 10.6) mm, rotated rx 0 ry 90 rz 0 deg; joints [-11.333, -27.468, 111.695, -15.329, -83.568, 50.752]
  Set speed (1000.0 mm/s)
  MoveL 4853 to (498.31, 492.3, 10.6) mm, rotated rx 0 ry 90 rz 0 deg; joints [-11.332, -27.467, 111.689, -15.328, -83.564, 50.753]
  Set speed (1000.0 mm/s)
  MoveL 4854 to (498.31, 493, 10.6) mm, rotated rx 0 ry 90 rz 0 deg; joints [-11.397, -27.464, 111.672, -15.394, -83.552, 50.763]
  Set speed (1000.0 mm/s)
  MoveL 4855 to (490.68, 490.68, 10.6) mm, rotated rx 0 ry 90 rz 0 deg; joints [-11.324, -27.602, 112.633, -15.297, -84.343, 50.538]
  Set speed (1000.0 mm/s)
  MoveL 4856 to (490.68, 490.68, 10.7) mm, rotated rx 0 ry 90 rz 0 deg; joints [-11.324, -27.613, 112.638, -15.298, -84.338, 50.539]
  Set speed (30.0 mm/s)
  Call Extruder(0.767)
  MoveL 4857 to (509.32, 509.32, 10.7) mm, rotated rx 0 ry 90 rz 0 deg; joints [-12.669, -27.201, 109.943, -16.726, -82.183, 51.312]
  MoveL 4858 to (509.44, 509.44, 10.7) mm, rotated rx 0 ry 90 rz 0 deg; joints [-12.677, -27.198, 109.925, -16.735, -82.169, 51.317]
  Set speed (120.0 mm/s)
  MoveL 4859 to (507.96, 501.93, 10.7) mm, rotated rx 0 ry 90 rz 0 deg; joints [-12.03, -27.26, 110.3, -16.07, -82.447, 51.15]
  Set speed (30.0 mm/s)
  Call Extruder(0.304)
  MoveL 4860 to (500.58, 509.32, 10.7) mm, rotated rx 0 ry 90 rz 0 deg; joints [-12.847, -27.37, 110.989, -16.873, -83.029, 51.077]
  Set speed (120.0 mm/s)
  MoveL 4861 to (499.42, 509.32, 10.7) mm, rotated rx 0 ry 90 rz 0 deg; joints [-12.872, -27.392, 111.127, -16.893, -83.142, 51.045]
  Set speed (30.0 mm/s)
  Call Extruder(0.360)
  MoveL 4862 to (490.68, 500.58, 10.7) mm, rotated rx 0 ry 90 rz 0 deg; joints [-12.247, -27.579, 112.394, -16.23, -84.158, 50.676]
  Set speed (120.0 mm/s)
  MoveL 4863 to (490.68, 499.42, 10.7) mm, rotated rx 0 ry 90 rz 0 deg; joints [-12.139, -27.583, 112.424, -16.121, -84.18, 50.659]
  Set speed (30.0 mm/s)
  Call Extruder(0.284)
  MoveL 4864 to (497.58, 492.52, 10.7) mm, rotated rx 0 ry 90 rz 0 deg; joints [-11.367, -27.49, 111.776, -15.361, -83.627, 50.739]
  MoveL 4865 to (497.7, 492.4, 10.7) mm, rotated rx 0 ry 90 rz 0 deg; joints [-11.353, -27.488, 111.764, -15.348, -83.617, 50.741]
  Set speed (120.0 mm/s)
  MoveL 4866 to (501.14, 492.33, 10.7) mm, rotated rx 0 ry 90 rz 0 deg; joints [-11.283, -27.427, 111.356, -15.288, -83.28, 50.826]
  Set speed (1000.0 mm/s)
  MoveL 4867 to (501.39, 491.49, 10.7) mm, rotated rx 0 ry 90 rz 0 deg; joints [-11.201, -27.425, 111.346, -15.206, -83.27, 50.82]
  Set speed (30.0 mm/s)
  Call Extruder(0.247)
  MoveL 4868 to (507.38, 497.49, 10.7) mm, rotated rx 0 ry 90 rz 0 deg; joints [-11.638, -27.29, 110.482, -15.67, -82.581, 51.063]
  MoveL 4869 to (507.51, 497.61, 10.7) mm, rotated rx 0 ry 90 rz 0 deg; joints [-11.647, -27.287, 110.464, -15.68, -82.567, 51.068]
  Set speed (120.0 mm/s)
  MoveL 4870 to (509.32, 490.68, 10.7) mm, rotated rx 0 ry 90 rz 0 deg; joints [-10.985, -27.278, 110.413, -15.014, -82.504, 51.003]
  Set speed (30.0 mm/s)
  Call Extruder(0.767)
  MoveL 4871 to (490.68, 509.32, 10.7) mm, rotated rx 0 ry 90 rz 0 deg; joints [-13.056, -27.546, 112.163, -17.05, -83.99, 50.804]
  MoveL 4872 to (490.56, 509.44, 10.7) mm, rotated rx 0 ry 90 rz 0 deg; joints [-13.07, -27.548, 112.174, -17.063, -83.999, 50.803]
  Set speed (120.0 mm/s)
  MoveL 4873 to (497.79, 492.37, 10.7) mm, rotated rx 0 ry 90 rz 0 deg; joints [-11.348, -27.487, 111.755, -15.343, -83.609, 50.742]
  Set speed (1000.0 mm/s)
  MoveL 4874 to (497.86, 492.3, 10.7) mm, rotated rx 0 ry 90 rz 0 deg; joints [-11.341, -27.486, 111.748, -15.336, -83.603, 50.743]
  Set speed (15.0 mm/s)
  Call Extruder(0.095)
  MoveL 4875 to (501.11, 492.3, 10.7) mm, rotated rx 0 ry 90 rz 0 deg; joints [-11.281, -27.427, 111.36, -15.285, -83.284, 50.825]
  Call Extruder(0.055)
  MoveL 4876 to (501.11, 490.4, 10.7) mm, rotated rx 0 ry 90 rz 0 deg; joints [-11.106, -27.434, 111.405, -15.109, -83.315, 50.797]
  Call Extruder(0.247)
  MoveL 4877 to (509.6, 490.4, 10.7) mm, rotated rx 0 ry 90 rz 0 deg; joints [-10.955, -27.274, 110.386, -14.984, -82.481, 51.005]
  Call Extruder(0.207)
  MoveL 4878 to (509.6, 497.51, 10.7) mm, rotated rx 0 ry 90 rz 0 deg; joints [-11.599, -27.246, 110.215, -15.639, -82.364, 51.119]
  Call Extruder(0.056)
  MoveL 4879 to (507.67, 497.51, 10.7) mm, rotated rx 0 ry 90 rz 0 deg; joints [-11.635, -27.284, 110.448, -15.668, -82.553, 51.07]
  Call Extruder(0.121)
  MoveL 4880 to (507.66, 501.65, 10.7) mm, rotated rx 0 ry 90 rz 0 deg; joints [-12.011, -27.267, 110.344, -16.049, -82.481, 51.138]
  Call Extruder(0.056)
  MoveL 4881 to (509.6, 501.66, 10.7) mm, rotated rx 0 ry 90 rz 0 deg; joints [-11.974, -27.229, 110.111, -16.019, -82.293, 51.188]
  Call Extruder(0.231)
  MoveL 4882 to (509.6, 509.6, 10.7) mm, rotated rx 0 ry 90 rz 0 deg; joints [-12.688, -27.194, 109.901, -16.747, -82.151, 51.324]
  Call Extruder(0.559)
  MoveL 4883 to (490.4, 509.6, 10.7) mm, rotated rx 0 ry 90 rz 0 deg; joints [-13.088, -27.55, 112.188, -17.081, -84.011, 50.801]
  MoveL 4884 to (490.4, 490.4, 10.7) mm, rotated rx 0 ry 90 rz 0 deg; joints [-11.303, -27.618, 112.678, -15.276, -84.371, 50.528]
  Call Extruder(0.217)
  MoveL 4885 to (497.86, 490.4, 10.7) mm, rotated rx 0 ry 90 rz 0 deg; joints [-11.165, -27.492, 111.793, -15.158, -83.636, 50.716]
  Call Extruder(0.055)
  MoveL 4886 to (497.86, 492.3, 10.7) mm, rotated rx 0 ry 90 rz 0 deg; joints [-11.341, -27.486, 111.748, -15.336, -83.603, 50.743]
  Set speed (120.0 mm/s)
  MoveL 4887 to (498.26, 492.3, 10.7) mm, rotated rx 0 ry 90 rz 0 deg; joints [-11.333, -27.479, 111.7, -15.329, -83.564, 50.753]
  Set speed (1000.0 mm/s)
  MoveL 4888 to (498.26, 493, 10.7) mm, rotated rx 0 ry 90 rz 0 deg; joints [-11.398, -27.476, 111.684, -15.395, -83.552, 50.763]
  Set speed (1000.0 mm/s)
  MoveL 4889 to (490.68, 490.68, 10.7) mm, rotated rx 0 ry 90 rz 0 deg; joints [-11.324, -27.613, 112.638, -15.298, -84.338, 50.539]
  Set speed (1000.0 mm/s)
  MoveL 4890 to (490.68, 490.68, 10.8) mm, rotated rx 0 ry 90 rz 0 deg; joints [-11.324, -27.624, 112.643, -15.298, -84.333, 50.541]
  Set speed (30.0 mm/s)
  Call Extruder(0.767)
  MoveL 4891 to (509.32, 509.32, 10.8) mm, rotated rx 0 ry 90 rz 0 deg; joints [-12.669, -27.212, 109.948, -16.726, -82.178, 51.313]
  MoveL 4892 to (509.44, 509.44, 10.8) mm, rotated rx 0 ry 90 rz 0 deg; joints [-12.677, -27.209, 109.93, -16.735, -82.164, 51.319]
  Set speed (120.0 mm/s)
  MoveL 4893 to (507.91, 501.99, 10.8) mm, rotated rx 0 ry 90 rz 0 deg; joints [-12.036, -27.271, 110.311, -16.077, -82.446, 51.151]
  Set speed (30.0 mm/s)
  Call Extruder(0.302)
  MoveL 4894 to (500.58, 509.32, 10.8) mm, rotated rx 0 ry 90 rz 0 deg; joints [-12.847, -27.381, 110.995, -16.873, -83.024, 51.078]
  Set speed (120.0 mm/s)
  MoveL 4895 to (499.42, 509.32, 10.8) mm, rotated rx 0 ry 90 rz 0 deg; joints [-12.872, -27.402, 111.133, -16.893, -83.137, 51.047]
  Set speed (30.0 mm/s)
  Call Extruder(0.360)
  MoveL 4896 to (490.68, 500.58, 10.8) mm, rotated rx 0 ry 90 rz 0 deg; joints [-12.247, -27.59, 112.399, -16.231, -84.153, 50.677]
  Set speed (120.0 mm/s)
  MoveL 4897 to (490.68, 499.42, 10.8) mm, rotated rx 0 ry 90 rz 0 deg; joints [-12.139, -27.594, 112.429, -16.122, -84.175, 50.661]
  Set speed (30.0 mm/s)
  Call Extruder(0.282)
  MoveL 4898 to (497.52, 492.58, 10.8) mm, rotated rx 0 ry 90 rz 0 deg; joints [-11.373, -27.501, 111.787, -15.367, -83.626, 50.74]
  MoveL 4899 to (497.64, 492.45, 10.8) mm, rotated rx 0 ry 90 rz 0 deg; joints [-11.359, -27.499, 111.775, -15.354, -83.616, 50.742]
  Set speed (120.0 mm/s)
  MoveL 4900 to (501.2, 492.33, 10.8) mm, rotated rx 0 ry 90 rz 0 deg; joints [-11.282, -27.436, 111.354, -15.287, -83.269, 50.829]
  Set speed (1000.0 mm/s)
  MoveL 4901 to (501.45, 491.55, 10.8) mm, rotated rx 0 ry 90 rz 0 deg; joints [-11.206, -27.434, 111.342, -15.211, -83.257, 50.824]
  Set speed (30.0 mm/s)
  Call Extruder(0.244)
  MoveL 4902 to (507.39, 497.49, 10.8) mm, rotated rx 0 ry 90 rz 0 deg; joints [-11.638, -27.3, 110.487, -15.67, -82.576, 51.064]
  MoveL 4903 to (507.51, 497.61, 10.8) mm, rotated rx 0 ry 90 rz 0 deg; joints [-11.647, -27.297, 110.469, -15.68, -82.562, 51.069]
  Set speed (120.0 mm/s)
  MoveL 4904 to (509.32, 490.68, 10.8) mm, rotated rx 0 ry 90 rz 0 deg; joints [-10.985, -27.289, 110.418, -15.014, -82.499, 51.004]
  Set speed (30.0 mm/s)
  Call Extruder(0.767)
  MoveL 4905 to (490.68, 509.32, 10.8) mm, rotated rx 0 ry 90 rz 0 deg; joints [-13.056, -27.557, 112.168, -17.05, -83.984, 50.806]
  MoveL 4906 to (490.56, 509.44, 10.8) mm, rotated rx 0 ry 90 rz 0 deg; joints [-13.07, -27.558, 112.179, -17.064, -83.994, 50.805]
  Set speed (120.0 mm/s)
  MoveL 4907 to (497.73, 492.37, 10.8) mm, rotated rx 0 ry 90 rz 0 deg; joints [-11.35, -27.498, 111.767, -15.345, -83.609, 50.742]
  Set speed (1000.0 mm/s)
  MoveL 4908 to (497.8, 492.3, 10.8) mm, rotated rx 0 ry 90 rz 0 deg; joints [-11.342, -27.497, 111.76, -15.337, -83.604, 50.743]
  Set speed (15.0 mm/s)
  Call Extruder(0.010)
  MoveL 4909 to (498.15, 492.3, 10.8) mm, rotated rx 0 ry 90 rz 0 deg; joints [-11.335, -27.491, 111.718, -15.331, -83.569, 50.752]
  Call Extruder(0.088)
  MoveL 4910 to (501.17, 492.3, 10.8) mm, rotated rx 0 ry 90 rz 0 deg; joints [-11.28, -27.437, 111.358, -15.285, -83.272, 50.828]
  Call Extruder(0.055)
  MoveL 4911 to (501.17, 490.4, 10.8) mm, rotated rx 0 ry 90 rz 0 deg; joints [-11.105, -27.444, 111.403, -15.108, -83.304, 50.8]
  Call Extruder(0.245)
  MoveL 4912 to (509.6, 490.4, 10.8) mm, rotated rx 0 ry 90 rz 0 deg; joints [-10.955, -27.285, 110.391, -14.984, -82.476, 51.007]
  Call Extruder(0.205)
  MoveL 4913 to (509.6, 497.45, 10.8) mm, rotated rx 0 ry 90 rz 0 deg; joints [-11.594, -27.257, 110.221, -15.633, -82.36, 51.12]
  Call Extruder(0.056)
  MoveL 4914 to (507.67, 497.45, 10.8) mm, rotated rx 0 ry 90 rz 0 deg; joints [-11.63, -27.295, 110.454, -15.663, -82.549, 51.071]
  Call Extruder(0.124)
  MoveL 4915 to (507.66, 501.71, 10.8) mm, rotated rx 0 ry 90 rz 0 deg; joints [-12.016, -27.277, 110.347, -16.055, -82.475, 51.14]
  Call Extruder(0.056)
  MoveL 4916 to (509.6, 501.71, 10.8) mm, rotated rx 0 ry 90 rz 0 deg; joints [-11.979, -27.239, 110.114, -16.025, -82.287, 51.19]
  Call Extruder(0.230)
  MoveL 4917 to (509.6, 509.6, 10.8) mm, rotated rx 0 ry 90 rz 0 deg; joints [-12.688, -27.205, 109.907, -16.747, -82.146, 51.326]
  Call Extruder(0.559)
  MoveL 4918 to (490.4, 509.6, 10.8) mm, rotated rx 0 ry 90 rz 0 deg; joints [-13.088, -27.56, 112.193, -17.081, -84.006, 50.803]
  MoveL 4919 to (490.4, 490.4, 10.8) mm, rotated rx 0 ry 90 rz 0 deg; joints [-11.303, -27.629, 112.683, -15.276, -84.365, 50.53]
  Call Extruder(0.205)
  MoveL 4920 to (497.45, 490.4, 10.8) mm, rotated rx 0 ry 90 rz 0 deg; joints [-11.173, -27.51, 111.847, -15.165, -83.67, 50.707]
  Call Extruder(0.010)
  MoveL 4921 to (497.8, 490.4, 10.8) mm, rotated rx 0 ry 90 rz 0 deg; joints [-11.166, -27.504, 111.805, -15.159, -83.636, 50.716]
  Call Extruder(0.007)
  MoveL 4922 to (497.8, 490.75, 10.8) mm, rotated rx 0 ry 90 rz 0 deg; joints [-11.199, -27.503, 111.797, -15.192, -83.63, 50.721]
  Call Extruder(0.035)
  MoveL 4923 to (497.8, 491.95, 10.8) mm, rotated rx 0 ry 90 rz 0 deg; joints [-11.31, -27.498, 111.768, -15.304, -83.61, 50.738]
  Call Extruder(0.007)
  MoveL 4924 to (497.8, 492.3, 10.8) mm, rotated rx 0 ry 90 rz 0 deg; joints [-11.342, -27.497, 111.76, -15.337, -83.604, 50.743]
  Set speed (120.0 mm/s)
  MoveL 4925 to (498.15, 492.3, 10.8) mm, rotated rx 0 ry 90 rz 0 deg; joints [-11.335, -27.491, 111.718, -15.331, -83.569, 50.752]
  Set speed (1000.0 mm/s)
  MoveL 4926 to (498.2, 492.3, 10.8) mm, rotated rx 0 ry 90 rz 0 deg; joints [-11.334, -27.49, 111.712, -15.331, -83.564, 50.753]
  Set speed (1000.0 mm/s)
  MoveL 4927 to (498.2, 493, 10.8) mm, rotated rx 0 ry 90 rz 0 deg; joints [-11.399, -27.488, 111.696, -15.396, -83.552, 50.763]
  Set speed (1000.0 mm/s)
  MoveL 4928 to (490.68, 490.68, 10.8) mm, rotated rx 0 ry 90 rz 0 deg; joints [-11.324, -27.624, 112.643, -15.298, -84.333, 50.541]
  Set speed (1000.0 mm/s)
  MoveL 4929 to (490.68, 490.68, 10.9) mm, rotated rx 0 ry 90 rz 0 deg; joints [-11.324, -27.634, 112.648, -15.298, -84.328, 50.542]
  Set speed (30.0 mm/s)
  Call Extruder(0.767)
  MoveL 4930 to (509.32, 509.32, 10.9) mm, rotated rx 0 ry 90 rz 0 deg; joints [-12.669, -27.222, 109.953, -16.726, -82.173, 51.315]
  MoveL 4931 to (509.44, 509.44, 10.9) mm, rotated rx 0 ry 90 rz 0 deg; joints [-12.677, -27.219, 109.935, -16.735, -82.159, 51.32]
  Set speed (120.0 mm/s)
  MoveL 4932 to (507.85, 502.05, 10.9) mm, rotated rx 0 ry 90 rz 0 deg; joints [-12.042, -27.283, 110.321, -16.083, -82.446, 51.152]
  Set speed (30.0 mm/s)
  Call Extruder(0.299)
  MoveL 4933 to (500.58, 509.32, 10.9) mm, rotated rx 0 ry 90 rz 0 deg; joints [-12.847, -27.391, 111, -16.873, -83.019, 51.08]
  Set speed (120.0 mm/s)
  MoveL 4934 to (499.42, 509.32, 10.9) mm, rotated rx 0 ry 90 rz 0 deg; joints [-12.872, -27.413, 111.138, -16.893, -83.131, 51.048]
  Set speed (30.0 mm/s)
  Call Extruder(0.360)
  MoveL 4935 to (490.68, 500.58, 10.9) mm, rotated rx 0 ry 90 rz 0 deg; joints [-12.247, -27.6, 112.404, -16.231, -84.148, 50.679]
  Set speed (120.0 mm/s)
  MoveL 4936 to (490.68, 499.42, 10.9) mm, rotated rx 0 ry 90 rz 0 deg; joints [-12.139, -27.604, 112.434, -16.122, -84.17, 50.662]
  Set speed (30.0 mm/s)
  Call Extruder(0.282)
  MoveL 4937 to (497.52, 492.58, 10.9) mm, rotated rx 0 ry 90 rz 0 deg; joints [-11.373, -27.512, 111.792, -15.368, -83.621, 50.742]
  MoveL 4938 to (497.64, 492.46, 10.9) mm, rotated rx 0 ry 90 rz 0 deg; joints [-11.359, -27.51, 111.78, -15.354, -83.611, 50.743]
  Set speed (120.0 mm/s)
  MoveL 4939 to (501.27, 492.33, 10.9) mm, rotated rx 0 ry 90 rz 0 deg; joints [-11.28, -27.446, 111.351, -15.286, -83.257, 50.832]
  Set speed (1000.0 mm/s)
  MoveL 4940 to (501.52, 491.62, 10.9) mm, rotated rx 0 ry 90 rz 0 deg; joints [-11.211, -27.444, 111.338, -15.216, -83.245, 50.828]
  Set speed (30.0 mm/s)
  Call Extruder(0.242)
  MoveL 4941 to (507.38, 497.49, 10.9) mm, rotated rx 0 ry 90 rz 0 deg; joints [-11.638, -27.311, 110.492, -15.67, -82.571, 51.066]
  MoveL 4942 to (507.51, 497.61, 10.9) mm, rotated rx 0 ry 90 rz 0 deg; joints [-11.647, -27.308, 110.475, -15.68, -82.556, 51.071]
  Set speed (120.0 mm/s)
  MoveL 4943 to (509.32, 490.68, 10.9) mm, rotated rx 0 ry 90 rz 0 deg; joints [-10.985, -27.299, 110.423, -15.014, -82.494, 51.005]
  Set speed (30.0 mm/s)
  Call Extruder(0.767)
  MoveL 4944 to (490.68, 509.32, 10.9) mm, rotated rx 0 ry 90 rz 0 deg; joints [-13.056, -27.567, 112.173, -17.05, -83.979, 50.808]
  MoveL 4945 to (490.56, 509.44, 10.9) mm, rotated rx 0 ry 90 rz 0 deg; joints [-13.07, -27.569, 112.184, -17.064, -83.989, 50.806]
  Set speed (120.0 mm/s)
  MoveL 4946 to (497.67, 492.37, 10.9) mm, rotated rx 0 ry 90 rz 0 deg; joints [-11.351, -27.51, 111.779, -15.346, -83.61, 50.743]
  Set speed (1000.0 mm/s)
  MoveL 4947 to (497.74, 492.3, 10.9) mm, rotated rx 0 ry 90 rz 0 deg; joints [-11.343, -27.509, 111.772, -15.338, -83.604, 50.743]
  Set speed (15.0 mm/s)
  Call Extruder(0.010)
  MoveL 4948 to (498.09, 492.3, 10.9) mm, rotated rx 0 ry 90 rz 0 deg; joints [-11.336, -27.503, 111.73, -15.332, -83.569, 50.752]
  Call Extruder(0.081)
  MoveL 4949 to (500.89, 492.3, 10.9) mm, rotated rx 0 ry 90 rz 0 deg; joints [-11.285, -27.453, 111.397, -15.289, -83.295, 50.822]
  Call Extruder(0.010)
  MoveL 4950 to (501.24, 492.3, 10.9) mm, rotated rx 0 ry 90 rz 0 deg; joints [-11.278, -27.446, 111.355, -15.284, -83.261, 50.831]
  Call Extruder(0.007)
  MoveL 4951 to (501.24, 491.95, 10.9) mm, rotated rx 0 ry 90 rz 0 deg; joints [-11.246, -27.447, 111.364, -15.251, -83.267, 50.826]
  Call Extruder(0.035)
  MoveL 4952 to (501.24, 490.75, 10.9) mm, rotated rx 0 ry 90 rz 0 deg; joints [-11.136, -27.452, 111.392, -15.14, -83.287, 50.808]
  Call Extruder(0.010)
  MoveL 4953 to (501.24, 490.4, 10.9) mm, rotated rx 0 ry 90 rz 0 deg; joints [-11.104, -27.453, 111.4, -15.107, -83.293, 50.803]
  Call Extruder(0.007)
  MoveL 4954 to (501.59, 490.4, 10.9) mm, rotated rx 0 ry 90 rz 0 deg; joints [-11.098, -27.447, 111.358, -15.102, -83.258, 50.812]
  Call Extruder(0.233)
  MoveL 4955 to (509.6, 490.4, 10.9) mm, rotated rx 0 ry 90 rz 0 deg; joints [-10.955, -27.295, 110.396, -14.984, -82.471, 51.008]
  Call Extruder(0.203)
  MoveL 4956 to (509.6, 497.39, 10.9) mm, rotated rx 0 ry 90 rz 0 deg; joints [-11.588, -27.268, 110.228, -15.628, -82.356, 51.12]
  Call Extruder(0.056)
  MoveL 4957 to (507.67, 497.39, 10.9) mm, rotated rx 0 ry 90 rz 0 deg; joints [-11.625, -27.306, 110.461, -15.657, -82.545, 51.071]
  Call Extruder(0.127)
  MoveL 4958 to (507.66, 501.77, 10.9) mm, rotated rx 0 ry 90 rz 0 deg; joints [-12.021, -27.288, 110.351, -16.06, -82.469, 51.143]
  Call Extruder(0.056)
  MoveL 4959 to (509.6, 501.77, 10.9) mm, rotated rx 0 ry 90 rz 0 deg; joints [-11.984, -27.249, 110.118, -16.03, -82.281, 51.193]
  Call Extruder(0.228)
  MoveL 4960 to (509.6, 509.6, 10.9) mm, rotated rx 0 ry 90 rz 0 deg; joints [-12.688, -27.215, 109.912, -16.747, -82.141, 51.327]
  Call Extruder(0.559)
  MoveL 4961 to (490.4, 509.6, 10.9) mm, rotated rx 0 ry 90 rz 0 deg; joints [-13.088, -27.571, 112.198, -17.081, -84.001, 50.804]
  MoveL 4962 to (490.4, 490.4, 10.9) mm, rotated rx 0 ry 90 rz 0 deg; joints [-11.303, -27.64, 112.688, -15.276, -84.36, 50.531]
  Call Extruder(0.204)
  MoveL 4963 to (497.39, 490.4, 10.9) mm, rotated rx 0 ry 90 rz 0 deg; joints [-11.174, -27.522, 111.858, -15.166, -83.671, 50.707]
  Call Extruder(0.010)
  MoveL 4964 to (497.74, 490.4, 10.9) mm, rotated rx 0 ry 90 rz 0 deg; joints [-11.167, -27.515, 111.817, -15.16, -83.636, 50.716]
  Call Extruder(0.007)
  MoveL 4965 to (497.75, 490.75, 10.9) mm, rotated rx 0 ry 90 rz 0 deg; joints [-11.2, -27.514, 111.809, -15.193, -83.63, 50.721]
  Call Extruder(0.035)
  MoveL 4966 to (497.74, 491.95, 10.9) mm, rotated rx 0 ry 90 rz 0 deg; joints [-11.311, -27.51, 111.78, -15.305, -83.61, 50.738]
  Call Extruder(0.007)
  MoveL 4967 to (497.74, 492.3, 10.9) mm, rotated rx 0 ry 90 rz 0 deg; joints [-11.343, -27.509, 111.772, -15.338, -83.604, 50.743]
  Set speed (120.0 mm/s)
  MoveL 4968 to (498.09, 492.3, 10.9) mm, rotated rx 0 ry 90 rz 0 deg; joints [-11.336, -27.503, 111.73, -15.332, -83.569, 50.752]
  Set speed (1000.0 mm/s)
  MoveL 4969 to (498.14, 492.3, 10.9) mm, rotated rx 0 ry 90 rz 0 deg; joints [-11.335, -27.502, 111.724, -15.332, -83.565, 50.753]
  Set speed (1000.0 mm/s)
  MoveL 4970 to (498.14, 493, 10.9) mm, rotated rx 0 ry 90 rz 0 deg; joints [-11.4, -27.499, 111.708, -15.397, -83.553, 50.763]
  Set speed (1000.0 mm/s)
  MoveL 4971 to (490.68, 490.68, 10.9) mm, rotated rx 0 ry 90 rz 0 deg; joints [-11.324, -27.634, 112.648, -15.298, -84.328, 50.542]
  Set speed (1000.0 mm/s)
  MoveL 4972 to (490.68, 490.68, 11) mm, rotated rx 0 ry 90 rz 0 deg; joints [-11.324, -27.645, 112.654, -15.298, -84.322, 50.544]
  Set speed (30.0 mm/s)
  Call Extruder(0.767)
  MoveL 4973 to (509.32, 509.32, 11) mm, rotated rx 0 ry 90 rz 0 deg; joints [-12.669, -27.232, 109.958, -16.726, -82.168, 51.317]
  MoveL 4974 to (509.44, 509.44, 11) mm, rotated rx 0 ry 90 rz 0 deg; joints [-12.677, -27.229, 109.94, -16.736, -82.154, 51.322]
  Set speed (120.0 mm/s)
  MoveL 4975 to (507.8, 502.1, 11) mm, rotated rx 0 ry 90 rz 0 deg; joints [-12.049, -27.294, 110.332, -16.089, -82.445, 51.153]
  Set speed (30.0 mm/s)
  Call Extruder(0.297)
  MoveL 4976 to (500.58, 509.32, 11) mm, rotated rx 0 ry 90 rz 0 deg; joints [-12.847, -27.402, 111.005, -16.873, -83.014, 51.081]
  Set speed (120.0 mm/s)
  MoveL 4977 to (499.42, 509.32, 11) mm, rotated rx 0 ry 90 rz 0 deg; joints [-12.872, -27.423, 111.143, -16.894, -83.126, 51.05]
  Set speed (30.0 mm/s)
  Call Extruder(0.360)
  MoveL 4978 to (490.68, 500.58, 11) mm, rotated rx 0 ry 90 rz 0 deg; joints [-12.247, -27.611, 112.41, -16.231, -84.143, 50.68]
  Set speed (120.0 mm/s)
  MoveL 4979 to (490.68, 499.42, 11) mm, rotated rx 0 ry 90 rz 0 deg; joints [-12.139, -27.615, 112.439, -16.122, -84.164, 50.664]
  Set speed (30.0 mm/s)
  Call Extruder(0.282)
  MoveL 4980 to (497.52, 492.58, 11) mm, rotated rx 0 ry 90 rz 0 deg; joints [-11.373, -27.522, 111.797, -15.368, -83.616, 50.743]
  MoveL 4981 to (497.64, 492.46, 11) mm, rotated rx 0 ry 90 rz 0 deg; joints [-11.359, -27.521, 111.785, -15.354, -83.606, 50.744]
  Set speed (120.0 mm/s)
  MoveL 4982 to (501.33, 492.33, 11) mm, rotated rx 0 ry 90 rz 0 deg; joints [-11.279, -27.455, 111.349, -15.285, -83.246, 50.835]
  Set speed (1000.0 mm/s)
  MoveL 4983 to (501.58, 491.68, 11) mm, rotated rx 0 ry 90 rz 0 deg; joints [-11.215, -27.453, 111.334, -15.221, -83.232, 50.832]
  Set speed (30.0 mm/s)
  Call Extruder(0.239)
  MoveL 4984 to (507.39, 497.49, 11) mm, rotated rx 0 ry 90 rz 0 deg; joints [-11.638, -27.321, 110.497, -15.671, -82.565, 51.067]
  MoveL 4985 to (507.51, 497.61, 11) mm, rotated rx 0 ry 90 rz 0 deg; joints [-11.647, -27.318, 110.48, -15.68, -82.551, 51.072]
  Set speed (120.0 mm/s)
  MoveL 4986 to (509.32, 490.68, 11) mm, rotated rx 0 ry 90 rz 0 deg; joints [-10.985, -27.31, 110.429, -15.014, -82.489, 51.007]
  Set speed (30.0 mm/s)
  Call Extruder(0.767)
  MoveL 4987 to (490.68, 509.32, 11) mm, rotated rx 0 ry 90 rz 0 deg; joints [-13.056, -27.578, 112.178, -17.05, -83.974, 50.809]
  MoveL 4988 to (490.56, 509.44, 11) mm, rotated rx 0 ry 90 rz 0 deg; joints [-13.07, -27.58, 112.189, -17.064, -83.984, 50.808]
  Set speed (120.0 mm/s)
  MoveL 4989 to (497.62, 492.37, 11) mm, rotated rx 0 ry 90 rz 0 deg; joints [-11.352, -27.521, 111.79, -15.347, -83.61, 50.743]
  Set speed (1000.0 mm/s)
  MoveL 4990 to (497.69, 492.3, 11) mm, rotated rx 0 ry 90 rz 0 deg; joints [-11.344, -27.52, 111.784, -15.339, -83.604, 50.743]
  Set speed (15.0 mm/s)
  Call Extruder(0.010)
  MoveL 4991 to (498.04, 492.3, 11) mm, rotated rx 0 ry 90 rz 0 deg; joints [-11.337, -27.514, 111.742, -15.333, -83.57, 50.752]
  Call Extruder(0.085)
  MoveL 4992 to (500.95, 492.3, 11) mm, rotated rx 0 ry 90 rz 0 deg; joints [-11.284, -27.462, 111.395, -15.288, -83.284, 50.825]
  Call Extruder(0.010)
  MoveL 4993 to (501.3, 492.3, 11) mm, rotated rx 0 ry 90 rz 0 deg; joints [-11.277, -27.456, 111.353, -15.283, -83.249, 50.834]
  Call Extruder(0.007)
  MoveL 4994 to (501.3, 491.95, 11) mm, rotated rx 0 ry 90 rz 0 deg; joints [-11.245, -27.457, 111.361, -15.25, -83.255, 50.829]
  Call Extruder(0.035)
  MoveL 4995 to (501.3, 490.75, 11) mm, rotated rx 0 ry 90 rz 0 deg; joints [-11.135, -27.461, 111.39, -15.139, -83.275, 50.811]
  Call Extruder(0.010)
  MoveL 4996 to (501.3, 490.4, 11) mm, rotated rx 0 ry 90 rz 0 deg; joints [-11.103, -27.462, 111.398, -15.106, -83.281, 50.806]
  Call Extruder(0.007)
  MoveL 4997 to (501.65, 490.4, 11) mm, rotated rx 0 ry 90 rz 0 deg; joints [-11.096, -27.456, 111.356, -15.101, -83.247, 50.815]
  Call Extruder(0.231)
  MoveL 4998 to (509.6, 490.4, 11) mm, rotated rx 0 ry 90 rz 0 deg; joints [-10.955, -27.305, 110.401, -14.984, -82.466, 51.009]
  Call Extruder(0.202)
  MoveL 4999 to (509.6, 497.33, 11) mm, rotated rx 0 ry 90 rz 0 deg; joints [-11.583, -27.278, 110.235, -15.623, -82.352, 51.121]
  Call Extruder(0.056)
  MoveL 5000 to (507.67, 497.33, 11) mm, rotated rx 0 ry 90 rz 0 deg; joints [-11.619, -27.316, 110.468, -15.652, -82.541, 51.072]
  Call Extruder(0.131)
  MoveL 5001 to (507.66, 501.82, 11) mm, rotated rx 0 ry 90 rz 0 deg; joints [-12.026, -27.298, 110.355, -16.066, -82.463, 51.145]
  Call Extruder(0.056)
  MoveL 5002 to (509.6, 501.83, 11) mm, rotated rx 0 ry 90 rz 0 deg; joints [-11.989, -27.26, 110.122, -16.036, -82.275, 51.195]
  Call Extruder(0.226)
  MoveL 5003 to (509.6, 509.6, 11) mm, rotated rx 0 ry 90 rz 0 deg; joints [-12.688, -27.226, 109.917, -16.747, -82.136, 51.329]
  Call Extruder(0.559)
  MoveL 5004 to (490.4, 509.6, 11) mm, rotated rx 0 ry 90 rz 0 deg; joints [-13.088, -27.582, 112.203, -17.082, -83.996, 50.806]
  MoveL 5005 to (490.4, 490.4, 11) mm, rotated rx 0 ry 90 rz 0 deg; joints [-11.303, -27.65, 112.693, -15.276, -84.355, 50.533]
  Call Extruder(0.202)
  MoveL 5006 to (497.34, 490.4, 11) mm, rotated rx 0 ry 90 rz 0 deg; joints [-11.175, -27.533, 111.87, -15.167, -83.671, 50.707]
  Call Extruder(0.010)
  MoveL 5007 to (497.69, 490.4, 11) mm, rotated rx 0 ry 90 rz 0 deg; joints [-11.168, -27.527, 111.829, -15.161, -83.637, 50.716]
  Call Extruder(0.007)
  MoveL 5008 to (497.69, 490.75, 11) mm, rotated rx 0 ry 90 rz 0 deg; joints [-11.201, -27.526, 111.82, -15.194, -83.631, 50.721]
  Call Extruder(0.035)
  MoveL 5009 to (497.69, 491.95, 11) mm, rotated rx 0 ry 90 rz 0 deg; joints [-11.312, -27.522, 111.792, -15.306, -83.61, 50.738]
  Call Extruder(0.007)
  MoveL 5010 to (497.69, 492.3, 11) mm, rotated rx 0 ry 90 rz 0 deg; joints [-11.344, -27.52, 111.784, -15.339, -83.604, 50.743]
  Set speed (120.0 mm/s)
  MoveL 5011 to (498.04, 492.3, 11) mm, rotated rx 0 ry 90 rz 0 deg; joints [-11.337, -27.514, 111.742, -15.333, -83.57, 50.752]
  Set speed (1000.0 mm/s)
  MoveL 5012 to (498.09, 492.3, 11) mm, rotated rx 0 ry 90 rz 0 deg; joints [-11.337, -27.513, 111.736, -15.333, -83.565, 50.753]
  Set speed (1000.0 mm/s)
  MoveL 5013 to (498.09, 493, 11) mm, rotated rx 0 ry 90 rz 0 deg; joints [-11.401, -27.511, 111.719, -15.398, -83.553, 50.764]
  Set speed (1000.0 mm/s)
  MoveL 5014 to (490.68, 490.68, 11) mm, rotated rx 0 ry 90 rz 0 deg; joints [-11.324, -27.645, 112.654, -15.298, -84.322, 50.544]
  Set speed (1000.0 mm/s)
  MoveL 5015 to (490.68, 490.68, 11.1) mm, rotated rx 0 ry 90 rz 0 deg; joints [-11.324, -27.656, 112.659, -15.298, -84.317, 50.545]
  Set speed (30.0 mm/s)
  Call Extruder(0.767)
  MoveL 5016 to (509.32, 509.32, 11.1) mm, rotated rx 0 ry 90 rz 0 deg; joints [-12.669, -27.243, 109.964, -16.726, -82.163, 51.318]
  MoveL 5017 to (509.44, 509.44, 11.1) mm, rotated rx 0 ry 90 rz 0 deg; joints [-12.677, -27.24, 109.945, -16.736, -82.149, 51.324]
  Set speed (120.0 mm/s)
  MoveL 5018 to (507.74, 502.16, 11.1) mm, rotated rx 0 ry 90 rz 0 deg; joints [-12.055, -27.306, 110.342, -16.095, -82.445, 51.154]
  Set speed (30.0 mm/s)
  Call Extruder(0.295)
  MoveL 5019 to (500.58, 509.32, 11.1) mm, rotated rx 0 ry 90 rz 0 deg; joints [-12.847, -27.412, 111.01, -16.874, -83.009, 51.083]
  Set speed (120.0 mm/s)
  MoveL 5020 to (499.42, 509.32, 11.1) mm, rotated rx 0 ry 90 rz 0 deg; joints [-12.872, -27.434, 111.148, -16.894, -83.121, 51.051]
  Set speed (30.0 mm/s)
  Call Extruder(0.360)
  MoveL 5021 to (490.68, 500.58, 11.1) mm, rotated rx 0 ry 90 rz 0 deg; joints [-12.247, -27.622, 112.415, -16.231, -84.138, 50.682]
  Set speed (120.0 mm/s)
  MoveL 5022 to (490.68, 499.42, 11.1) mm, rotated rx 0 ry 90 rz 0 deg; joints [-12.139, -27.626, 112.445, -16.122, -84.159, 50.665]
  Set speed (30.0 mm/s)
  Call Extruder(0.282)
  MoveL 5023 to (497.52, 492.58, 11.1) mm, rotated rx 0 ry 90 rz 0 deg; joints [-11.373, -27.533, 111.802, -15.368, -83.611, 50.745]
  MoveL 5024 to (497.64, 492.45, 11.1) mm, rotated rx 0 ry 90 rz 0 deg; joints [-11.359, -27.531, 111.791, -15.354, -83.601, 50.746]
  Set speed (120.0 mm/s)
  MoveL 5025 to (501.39, 492.33, 11.1) mm, rotated rx 0 ry 90 rz 0 deg; joints [-11.278, -27.464, 111.346, -15.284, -83.235, 50.838]
  Set speed (1000.0 mm/s)
  MoveL 5026 to (501.64, 491.74, 11.1) mm, rotated rx 0 ry 90 rz 0 deg; joints [-11.22, -27.462, 111.33, -15.226, -83.22, 50.836]
  Set speed (30.0 mm/s)
  Call Extruder(0.236)
  MoveL 5027 to (507.39, 497.49, 11.1) mm, rotated rx 0 ry 90 rz 0 deg; joints [-11.638, -27.332, 110.503, -15.671, -82.56, 51.069]
  MoveL 5028 to (507.51, 497.61, 11.1) mm, rotated rx 0 ry 90 rz 0 deg; joints [-11.647, -27.329, 110.485, -15.68, -82.546, 51.074]
  Set speed (120.0 mm/s)
  MoveL 5029 to (509.32, 490.68, 11.1) mm, rotated rx 0 ry 90 rz 0 deg; joints [-10.985, -27.32, 110.434, -15.014, -82.484, 51.008]
  Set speed (30.0 mm/s)
  Call Extruder(0.767)
  MoveL 5030 to (490.68, 509.32, 11.1) mm, rotated rx 0 ry 90 rz 0 deg; joints [-13.056, -27.589, 112.184, -17.05, -83.969, 50.811]
  MoveL 5031 to (490.56, 509.44, 11.1) mm, rotated rx 0 ry 90 rz 0 deg; joints [-13.07, -27.59, 112.195, -17.064, -83.978, 50.809]
  Set speed (120.0 mm/s)
  MoveL 5032 to (497.56, 492.37, 11.1) mm, rotated rx 0 ry 90 rz 0 deg; joints [-11.353, -27.533, 111.802, -15.348, -83.61, 50.743]
  Set speed (1000.0 mm/s)
  MoveL 5033 to (497.63, 492.3, 11.1) mm, rotated rx 0 ry 90 rz 0 deg; joints [-11.345, -27.532, 111.796, -15.34, -83.605, 50.743]
  Set speed (15.0 mm/s)
  Call Extruder(0.010)
  MoveL 5034 to (497.98, 492.3, 11.1) mm, rotated rx 0 ry 90 rz 0 deg; joints [-11.338, -27.526, 111.754, -15.335, -83.57, 50.752]
  Call Extruder(0.098)
  MoveL 5035 to (501.37, 492.3, 11.1) mm, rotated rx 0 ry 90 rz 0 deg; joints [-11.276, -27.465, 111.35, -15.282, -83.238, 50.837]
  Call Extruder(0.055)
  MoveL 5036 to (501.37, 490.4, 11.1) mm, rotated rx 0 ry 90 rz 0 deg; joints [-11.102, -27.472, 111.395, -15.105, -83.27, 50.809]
  Call Extruder(0.240)
  MoveL 5037 to (509.6, 490.4, 11.1) mm, rotated rx 0 ry 90 rz 0 deg; joints [-10.955, -27.316, 110.406, -14.985, -82.461, 51.011]
  Call Extruder(0.200)
  MoveL 5038 to (509.6, 497.27, 11.1) mm, rotated rx 0 ry 90 rz 0 deg; joints [-11.578, -27.289, 110.241, -15.617, -82.348, 51.121]
  Call Extruder(0.056)
  MoveL 5039 to (507.67, 497.27, 11.1) mm, rotated rx 0 ry 90 rz 0 deg; joints [-11.614, -27.327, 110.474, -15.647, -82.536, 51.072]
  Call Extruder(0.062)
  MoveL 5040 to (507.67, 499.41, 11.1) mm, rotated rx 0 ry 90 rz 0 deg; joints [-11.807, -27.318, 110.421, -15.844, -82.5, 51.107]
  Call Extruder(0.072)
  MoveL 5041 to (507.66, 501.88, 11.1) mm, rotated rx 0 ry 90 rz 0 deg; joints [-12.031, -27.308, 110.359, -16.071, -82.457, 51.148]
  Call Extruder(0.056)
  MoveL 5042 to (509.6, 501.88, 11.1) mm, rotated rx 0 ry 90 rz 0 deg; joints [-11.994, -27.27, 110.125, -16.041, -82.269, 51.198]
  Call Extruder(0.225)
  MoveL 5043 to (509.6, 509.6, 11.1) mm, rotated rx 0 ry 90 rz 0 deg; joints [-12.688, -27.236, 109.922, -16.748, -82.131, 51.331]
  Call Extruder(0.559)
  MoveL 5044 to (490.4, 509.6, 11.1) mm, rotated rx 0 ry 90 rz 0 deg; joints [-13.088, -27.592, 112.209, -17.082, -83.99, 50.807]
  MoveL 5045 to (490.4, 490.4, 11.1) mm, rotated rx 0 ry 90 rz 0 deg; joints [-11.303, -27.661, 112.698, -15.276, -84.35, 50.534]
  Call Extruder(0.210)
  MoveL 5046 to (497.63, 490.4, 11.1) mm, rotated rx 0 ry 90 rz 0 deg; joints [-11.169, -27.539, 111.841, -15.162, -83.637, 50.716]
  Call Extruder(0.045)
  MoveL 5047 to (497.63, 491.95, 11.1) mm, rotated rx 0 ry 90 rz 0 deg; joints [-11.313, -27.533, 111.804, -15.307, -83.611, 50.738]
  Call Extruder(0.007)
  MoveL 5048 to (497.63, 492.3, 11.1) mm, rotated rx 0 ry 90 rz 0 deg; joints [-11.345, -27.532, 111.796, -15.34, -83.605, 50.743]
  Set speed (120.0 mm/s)
  MoveL 5049 to (497.98, 492.3, 11.1) mm, rotated rx 0 ry 90 rz 0 deg; joints [-11.338, -27.526, 111.754, -15.335, -83.57, 50.752]
  Set speed (1000.0 mm/s)
  MoveL 5050 to (498.03, 492.3, 11.1) mm, rotated rx 0 ry 90 rz 0 deg; joints [-11.338, -27.525, 111.748, -15.334, -83.565, 50.753]
  Set speed (1000.0 mm/s)
  MoveL 5051 to (498.03, 493, 11.1) mm, rotated rx 0 ry 90 rz 0 deg; joints [-11.402, -27.522, 111.731, -15.399, -83.553, 50.764]
  Set speed (1000.0 mm/s)
  MoveL 5052 to (490.68, 490.68, 11.1) mm, rotated rx 0 ry 90 rz 0 deg; joints [-11.324, -27.656, 112.659, -15.298, -84.317, 50.545]
  Set speed (1000.0 mm/s)
  MoveL 5053 to (490.68, 490.68, 11.2) mm, rotated rx 0 ry 90 rz 0 deg; joints [-11.324, -27.666, 112.664, -15.298, -84.312, 50.546]
  Set speed (30.0 mm/s)
  Call Extruder(0.767)
  MoveL 5054 to (509.32, 509.32, 11.2) mm, rotated rx 0 ry 90 rz 0 deg; joints [-12.669, -27.253, 109.969, -16.727, -82.158, 51.32]
  MoveL 5055 to (509.44, 509.44, 11.2) mm, rotated rx 0 ry 90 rz 0 deg; joints [-12.677, -27.25, 109.951, -16.736, -82.144, 51.325]
  Set speed (120.0 mm/s)
  MoveL 5056 to (507.68, 502.21, 11.2) mm, rotated rx 0 ry 90 rz 0 deg; joints [-12.061, -27.317, 110.353, -16.102, -82.444, 51.155]
  Set speed (30.0 mm/s)
  Call Extruder(0.292)
  MoveL 5057 to (500.58, 509.32, 11.2) mm, rotated rx 0 ry 90 rz 0 deg; joints [-12.847, -27.423, 111.015, -16.874, -83.004, 51.085]
  Set speed (120.0 mm/s)
  MoveL 5058 to (499.42, 509.32, 11.2) mm, rotated rx 0 ry 90 rz 0 deg; joints [-12.872, -27.444, 111.153, -16.894, -83.116, 51.053]
  Set speed (30.0 mm/s)
  Call Extruder(0.360)
  MoveL 5059 to (490.68, 500.58, 11.2) mm, rotated rx 0 ry 90 rz 0 deg; joints [-12.247, -27.632, 112.42, -16.231, -84.132, 50.683]
  Set speed (120.0 mm/s)
  MoveL 5060 to (490.68, 499.42, 11.2) mm, rotated rx 0 ry 90 rz 0 deg; joints [-12.139, -27.636, 112.45, -16.122, -84.154, 50.667]
  Set speed (30.0 mm/s)
  Call Extruder(0.282)
  MoveL 5061 to (497.52, 492.58, 11.2) mm, rotated rx 0 ry 90 rz 0 deg; joints [-11.373, -27.544, 111.807, -15.368, -83.605, 50.746]
  MoveL 5062 to (497.64, 492.46, 11.2) mm, rotated rx 0 ry 90 rz 0 deg; joints [-11.359, -27.542, 111.796, -15.355, -83.595, 50.747]
  Set speed (120.0 mm/s)
  MoveL 5063 to (501.46, 492.33, 11.2) mm, rotated rx 0 ry 90 rz 0 deg; joints [-11.277, -27.474, 111.344, -15.284, -83.223, 50.841]
  Set speed (1000.0 mm/s)
  MoveL 5064 to (501.71, 491.81, 11.2) mm, rotated rx 0 ry 90 rz 0 deg; joints [-11.225, -27.471, 111.326, -15.232, -83.207, 50.84]
  Set speed (30.0 mm/s)
  Call Extruder(0.234)
  MoveL 5065 to (507.38, 497.49, 11.2) mm, rotated rx 0 ry 90 rz 0 deg; joints [-11.638, -27.342, 110.508, -15.671, -82.555, 51.07]
  MoveL 5066 to (507.51, 497.61, 11.2) mm, rotated rx 0 ry 90 rz 0 deg; joints [-11.647, -27.339, 110.49, -15.68, -82.541, 51.075]
  Set speed (120.0 mm/s)
  MoveL 5067 to (509.32, 490.68, 11.2) mm, rotated rx 0 ry 90 rz 0 deg; joints [-10.985, -27.331, 110.439, -15.015, -82.479, 51.01]
  Set speed (30.0 mm/s)
  Call Extruder(0.767)
  MoveL 5068 to (490.68, 509.32, 11.2) mm, rotated rx 0 ry 90 rz 0 deg; joints [-13.056, -27.599, 112.189, -17.05, -83.964, 50.812]
  MoveL 5069 to (490.56, 509.44, 11.2) mm, rotated rx 0 ry 90 rz 0 deg; joints [-13.07, -27.601, 112.2, -17.064, -83.973, 50.811]
  Set speed (120.0 mm/s)
  MoveL 5070 to (497.51, 492.37, 11.2) mm, rotated rx 0 ry 90 rz 0 deg; joints [-11.354, -27.545, 111.814, -15.349, -83.611, 50.743]
  Set speed (1000.0 mm/s)
  MoveL 5071 to (497.58, 492.3, 11.2) mm, rotated rx 0 ry 90 rz 0 deg; joints [-11.346, -27.544, 111.808, -15.341, -83.605, 50.743]
  Set speed (15.0 mm/s)
  Call Extruder(0.010)
  MoveL 5072 to (497.93, 492.3, 11.2) mm, rotated rx 0 ry 90 rz 0 deg; joints [-11.34, -27.537, 111.766, -15.336, -83.571, 50.752]
  Call Extruder(0.102)
  MoveL 5073 to (501.43, 492.3, 11.2) mm, rotated rx 0 ry 90 rz 0 deg; joints [-11.275, -27.474, 111.348, -15.281, -83.226, 50.84]
  Call Extruder(0.055)
  MoveL 5074 to (501.43, 490.4, 11.2) mm, rotated rx 0 ry 90 rz 0 deg; joints [-11.1, -27.481, 111.393, -15.105, -83.258, 50.812]
  Call Extruder(0.238)
  MoveL 5075 to (509.6, 490.4, 11.2) mm, rotated rx 0 ry 90 rz 0 deg; joints [-10.955, -27.326, 110.412, -14.985, -82.456, 51.012]
  Call Extruder(0.198)
  MoveL 5076 to (509.6, 497.21, 11.2) mm, rotated rx 0 ry 90 rz 0 deg; joints [-11.572, -27.3, 110.248, -15.612, -82.344, 51.122]
  Call Extruder(0.056)
  MoveL 5077 to (507.67, 497.21, 11.2) mm, rotated rx 0 ry 90 rz 0 deg; joints [-11.608, -27.338, 110.481, -15.641, -82.532, 51.073]
  Call Extruder(0.066)
  MoveL 5078 to (507.67, 499.46, 11.2) mm, rotated rx 0 ry 90 rz 0 deg; joints [-11.812, -27.329, 110.425, -15.849, -82.494, 51.109]
  Call Extruder(0.072)
  MoveL 5079 to (507.66, 501.94, 11.2) mm, rotated rx 0 ry 90 rz 0 deg; joints [-12.036, -27.318, 110.362, -16.076, -82.451, 51.15]
  Call Extruder(0.056)
  MoveL 5080 to (509.6, 501.94, 11.2) mm, rotated rx 0 ry 90 rz 0 deg; joints [-11.999, -27.28, 110.129, -16.046, -82.262, 51.2]
  Call Extruder(0.223)
